C05533=1107.470,43.607,-54.704,179.966,7.215,149.356
C05534=1107.464,43.857,-54.721,179.966,7.219,149.357
C05535=1107.459,44.106,-54.737,179.968,7.222,149.357
C05536=1107.455,44.355,-54.754,179.969,7.227,149.358
C05537=1107.449,44.605,-54.770,179.970,7.231,149.359
C05538=1107.444,44.855,-54.787,179.970,7.235,149.359
C05539=1107.440,45.104,-54.804,179.971,7.239,149.360
C05540=1107.435,45.353,-54.820,179.973,7.243,149.360
C05541=1107.430,45.602,-54.837,179.974,7.247,149.361
C05542=1107.425,45.852,-54.854,179.974,7.251,149.362
C05543=1107.420,46.101,-54.870,179.975,7.255,149.362
C05544=1107.415,46.351,-54.886,179.976,7.259,149.363
C05545=1107.411,46.601,-54.903,179.978,7.263,149.364
C05546=1107.405,46.850,-54.920,179.978,7.267,149.364
C05547=1107.400,47.099,-54.936,179.980,7.271,149.365
C05548=1107.396,47.349,-54.953,179.981,7.275,149.365
C05549=1107.390,47.598,-54.970,179.982,7.279,149.366
C05550=1107.385,47.847,-54.987,179.983,7.283,149.367
C05551=1107.381,48.097,-55.003,179.984,7.287,149.367
C05552=1107.375,48.346,-55.020,179.985,7.291,149.368
C05553=1107.371,48.595,-55.037,179.986,7.295,149.368
C05554=1107.366,48.845,-55.054,179.987,7.299,149.369
C05555=1107.361,49.094,-55.071,179.988,7.303,149.370
C05556=1107.356,49.343,-55.087,179.989,7.307,149.370
C05557=1107.351,49.593,-55.104,179.991,7.311,149.371
C05558=1107.347,49.806,-55.118,179.992,7.314,149.371
C05559=1107.343,50.020,-55.133,179.992,7.318,149.372
C05560=1107.338,50.235,-55.147,179.993,7.321,149.372
C05561=1107.334,50.448,-55.161,179.994,7.325,149.373
C05562=1107.330,50.662,-55.176,179.995,7.328,149.373
C05563=1107.326,50.876,-55.191,179.996,7.332,149.374
C05564=1107.322,51.090,-55.205,179.997,7.335,149.374
C05565=1107.318,51.304,-55.220,179.998,7.339,149.375
C05566=1107.312,51.553,-55.237,179.999,7.342,149.375
C05567=1107.308,51.803,-55.254,180.000,7.346,149.376
C05568=1107.302,52.052,-55.270,-179.999,7.350,149.376
C05569=1107.298,52.301,-55.287,-179.997,7.355,149.377
C05570=1107.293,52.551,-55.304,-179.997,7.358,149.378
C05571=1107.288,52.801,-55.321,-179.995,7.362,149.378
C05572=1107.284,53.050,-55.338,-179.994,7.366,149.379
C05573=1107.278,53.299,-55.355,-179.993,7.370,149.379
C05574=1107.274,53.548,-55.372,-179.992,7.374,149.380
C05575=1107.268,53.798,-55.389,-179.991,7.378,149.381
C05576=1107.264,54.047,-55.406,-179.990,7.382,149.381
C05577=1107.258,54.296,-55.424,-179.989,7.386,149.382
C05578=1107.254,54.545,-55.440,-179.987,7.390,149.382
C05579=1107.249,54.795,-55.458,-179.986,7.394,149.383
C05580=1107.244,55.045,-55.474,-179.985,7.398,149.383
C05581=1107.239,55.294,-55.491,-179.984,7.402,149.384
C05582=1107.235,55.543,-55.509,-179.983,7.406,149.384
C05583=1107.229,55.792,-55.526,-179.981,7.410,149.385
C05584=1107.224,56.042,-55.543,-179.981,7.414,149.386
C05585=1107.220,56.291,-55.560,-179.980,7.418,149.386
C05586=1107.214,56.541,-55.578,-179.978,7.422,149.387
C05587=1107.210,56.790,-55.594,-179.977,7.426,149.387
C05588=1107.205,57.040,-55.612,-179.975,7.430,149.388
C05589=1107.200,57.288,-55.629,-179.975,7.433,149.388
C05590=1107.195,57.538,-55.646,-179.973,7.437,149.389
C05591=1107.190,57.787,-55.664,-179.972,7.442,149.389
C05592=1107.185,58.037,-55.681,-179.971,7.446,149.390
C05593=1107.180,58.287,-55.698,-179.970,7.450,149.391
C05594=1107.176,58.535,-55.715,-179.969,7.453,149.391
C05595=1107.171,58.785,-55.732,-179.968,7.457,149.392
C05596=1107.165,59.035,-55.750,-179.966,7.461,149.392
C05597=1107.161,59.284,-55.767,-179.965,7.465,149.393
C05598=1107.155,59.533,-55.784,-179.963,7.469,149.393
C05599=1107.151,59.782,-55.802,-179.963,7.473,149.394
C05600=1107.146,60.032,-55.819,-179.961,7.477,149.394
C05601=1107.141,60.281,-55.837,-179.960,7.481,149.395
C05602=1107.136,60.531,-55.854,-179.959,7.485,149.395
C05603=1107.132,60.780,-55.871,-179.958,7.489,149.396
C05604=1107.127,61.029,-55.889,-179.956,7.493,149.396
C05605=1107.122,61.278,-55.907,-179.956,7.497,149.397
C05606=1107.117,61.528,-55.923,-179.954,7.501,149.397
C05607=1107.112,61.777,-55.941,-179.953,7.505,149.398
C05608=1107.107,62.027,-55.958,-179.951,7.509,149.399
C05609=1107.102,62.276,-55.976,-179.950,7.513,149.399
C05610=1107.098,62.526,-55.993,-179.949,7.516,149.400
C05611=1107.093,62.775,-56.011,-179.948,7.520,149.400
C05612=1107.087,63.025,-56.028,-179.947,7.524,149.401
C05613=1107.083,63.274,-56.046,-179.945,7.528,149.401
C05614=1107.079,63.487,-56.061,-179.944,7.531,149.402
C05615=1107.074,63.701,-56.076,-179.944,7.535,149.402
C05616=1107.070,63.915,-56.091,-179.942,7.539,149.403
C05617=1107.065,64.129,-56.106,-179.941,7.542,149.403
C05618=1107.062,64.342,-56.121,-179.940,7.545,149.404
C05619=1107.058,64.556,-56.136,-179.939,7.549,149.404
C05620=1107.054,64.770,-56.151,-179.938,7.552,149.404
C05621=1107.049,64.983,-56.167,-179.937,7.555,149.405
C05622=1107.044,65.233,-56.184,-179.935,7.559,149.405
C05623=1107.039,65.482,-56.202,-179.934,7.563,149.406
C05624=1107.035,65.731,-56.219,-179.933,7.567,149.406
C05625=1107.030,65.981,-56.236,-179.931,7.572,149.407
C05626=1107.025,66.230,-56.254,-179.930,7.575,149.407
C05627=1107.020,66.479,-56.272,-179.929,7.579,149.408
C05628=1107.015,66.729,-56.290,-179.928,7.583,149.409
C05629=1107.010,66.978,-56.308,-179.926,7.587,149.409
C05630=1107.006,67.228,-56.325,-179.925,7.591,149.410
C05631=1107.001,67.477,-56.343,-179.924,7.595,149.410
C05632=1106.996,67.726,-56.361,-179.923,7.598,149.411
C05633=1106.991,67.976,-56.379,-179.921,7.602,149.411
C05634=1106.986,68.225,-56.397,-179.920,7.606,149.412
C05635=1106.981,68.474,-56.415,-179.918,7.610,149.412
C05636=1106.976,68.724,-56.433,-179.917,7.615,149.413
C05637=1106.971,68.973,-56.451,-179.916,7.618,149.413
C05638=1106.966,69.223,-56.468,-179.915,7.623,149.414
C05639=1106.961,69.472,-56.486,-179.913,7.627,149.414
C05640=1106.956,69.721,-56.504,-179.912,7.630,149.415
C05641=1106.952,69.970,-56.521,-179.911,7.634,149.415
C05642=1106.947,70.219,-56.539,-179.909,7.638,149.416
C05643=1106.943,70.469,-56.557,-179.908,7.642,149.416
C05644=1106.938,70.718,-56.575,-179.907,7.646,149.417
C05645=1106.933,70.967,-56.593,-179.905,7.650,149.417
C05646=1106.928,71.216,-56.611,-179.904,7.654,149.418
C05647=1106.923,71.466,-56.629,-179.902,7.658,149.418
C05648=1106.918,71.715,-56.647,-179.901,7.661,149.419
C05649=1106.913,71.965,-56.665,-179.900,7.665,149.419
C05650=1106.908,72.214,-56.683,-179.899,7.669,149.420
C05651=1106.904,72.464,-56.701,-179.897,7.673,149.420
C05652=1106.899,72.713,-56.719,-179.896,7.677,149.421
C05653=1106.894,72.962,-56.737,-179.894,7.682,149.421
C05654=1106.889,73.211,-56.755,-179.893,7.685,149.422
C05655=1106.884,73.461,-56.773,-179.891,7.689,149.422
C05656=1106.879,73.710,-56.791,-179.890,7.693,149.423
C05657=1106.874,73.960,-56.810,-179.889,7.697,149.423
C05658=1106.870,74.209,-56.828,-179.888,7.701,149.424
C05659=1106.865,74.458,-56.846,-179.886,7.705,149.424
C05660=1106.860,74.707,-56.864,-179.885,7.709,149.425
C05661=1106.855,74.956,-56.882,-179.883,7.713,149.425
C05662=1106.851,75.206,-56.901,-179.882,7.717,149.426
C05663=1106.846,75.455,-56.919,-179.880,7.721,149.426
C05664=1106.841,75.704,-56.937,-179.879,7.725,149.427
C05665=1106.836,75.953,-56.955,-179.878,7.729,149.427
C05666=1106.830,76.203,-56.973,-179.876,7.733,149.428
C05667=1106.826,76.453,-56.992,-179.875,7.736,149.428
C05668=1106.821,76.701,-57.010,-179.874,7.740,149.429
C05669=1106.817,76.950,-57.028,-179.872,7.744,149.429
C05670=1106.812,77.164,-57.044,-179.871,7.747,149.430
C05671=1106.808,77.378,-57.059,-179.871,7.751,149.430
C05672=1106.804,77.592,-57.075,-179.870,7.754,149.431
C05673=1106.800,77.806,-57.091,-179.869,7.757,149.431
C05674=1106.796,78.019,-57.106,-179.868,7.760,149.432
C05675=1106.792,78.232,-57.122,-179.867,7.763,149.432
C05676=1106.788,78.446,-57.138,-179.867,7.766,149.433
C05677=1106.783,78.660,-57.154,-179.866,7.770,149.433
C05678=1106.779,78.910,-57.172,-179.864,7.773,149.434
C05679=1106.773,79.159,-57.191,-179.864,7.777,149.434
C05680=1106.769,79.408,-57.209,-179.862,7.781,149.435
C05681=1106.764,79.657,-57.228,-179.861,7.784,149.435
C05682=1106.760,79.907,-57.246,-179.860,7.789,149.436
C05683=1106.755,80.156,-57.264,-179.859,7.792,149.436
C05684=1106.749,80.405,-57.282,-179.858,7.796,149.437
C05685=1106.745,80.655,-57.302,-179.857,7.799,149.437
C05686=1106.740,80.904,-57.320,-179.856,7.803,149.438
C05687=1106.735,81.153,-57.338,-179.855,7.807,149.439
C05688=1106.730,81.402,-57.357,-179.854,7.811,149.439
C05689=1106.726,81.652,-57.375,-179.853,7.814,149.440
C05690=1106.721,81.901,-57.393,-179.852,7.818,149.440
C05691=1106.715,82.150,-57.412,-179.851,7.821,149.441
C05692=1106.711,82.400,-57.431,-179.850,7.826,149.441
C05693=1106.706,82.648,-57.449,-179.849,7.829,149.442
C05694=1106.702,82.897,-57.467,-179.848,7.833,149.442
C05695=1106.696,83.148,-57.486,-179.846,7.837,149.443
C05696=1106.692,83.396,-57.505,-179.846,7.840,149.444
C05697=1106.687,83.645,-57.523,-179.844,7.844,149.444
C05698=1106.682,83.895,-57.543,-179.844,7.848,149.445
C05699=1106.677,84.144,-57.561,-179.842,7.852,149.445
C05700=1106.673,84.394,-57.579,-179.841,7.855,149.446
C05701=1106.668,84.643,-57.598,-179.840,7.859,149.446
C05702=1106.663,84.892,-57.616,-179.839,7.863,149.447
C05703=1106.658,85.142,-57.636,-179.838,7.866,149.447
C05704=1106.653,85.391,-57.654,-179.837,7.871,149.448
C05705=1106.648,85.639,-57.673,-179.835,7.875,149.448
C05706=1106.643,85.890,-57.692,-179.834,7.878,149.449
C05707=1106.639,86.138,-57.710,-179.833,7.882,149.449
C05708=1106.635,86.388,-57.729,-179.832,7.885,149.450
C05709=1106.629,86.637,-57.748,-179.831,7.889,149.450
C05710=1106.625,86.885,-57.767,-179.829,7.893,149.451
C05711=1106.620,87.136,-57.786,-179.828,7.896,149.451
C05712=1106.615,87.384,-57.804,-179.827,7.901,149.452
C05713=1106.610,87.634,-57.823,-179.826,7.905,149.452
C05714=1106.605,87.883,-57.842,-179.825,7.908,149.453
C05715=1106.600,88.132,-57.860,-179.823,7.912,149.454
C05716=1106.596,88.382,-57.880,-179.822,7.916,149.454
C05717=1106.591,88.630,-57.898,-179.821,7.919,149.455
C05718=1106.586,88.880,-57.917,-179.820,7.923,149.455
C05719=1106.581,89.129,-57.936,-179.818,7.927,149.455
C05720=1106.577,89.378,-57.956,-179.818,7.931,149.456
C05721=1106.572,89.628,-57.973,-179.816,7.934,149.457
C05722=1106.567,89.877,-57.993,-179.814,7.938,149.457
C05723=1106.562,90.126,-58.012,-179.814,7.942,149.458
C05724=1106.557,90.376,-58.031,-179.812,7.946,149.458
C05725=1106.553,90.624,-58.049,-179.811,7.950,149.459
C05726=1106.548,90.839,-58.066,-179.810,7.953,149.459
C05727=1106.544,91.052,-58.083,-179.809,7.956,149.459
C05728=1106.540,91.266,-58.099,-179.808,7.959,149.460
C05729=1106.536,91.479,-58.114,-179.806,7.963,149.460
C05730=1106.532,91.693,-58.131,-179.805,7.966,149.461
C05731=1106.528,91.906,-58.147,-179.804,7.969,149.461
C05732=1106.523,92.120,-58.164,-179.803,7.972,149.462
C05733=1106.520,92.334,-58.181,-179.802,7.975,149.462
C05734=1106.515,92.582,-58.199,-179.801,7.979,149.462
C05735=1106.510,92.833,-58.218,-179.799,7.983,149.463
C05736=1106.505,93.082,-58.237,-179.798,7.987,149.463
C05737=1106.501,93.331,-58.256,-179.797,7.990,149.464
C05738=1106.495,93.580,-58.276,-179.795,7.994,149.464
C05739=1106.491,93.829,-58.295,-179.794,7.998,149.465
C05740=1106.486,94.078,-58.313,-179.793,8.001,149.465
C05741=1106.481,94.328,-58.333,-179.791,8.005,149.466
C05742=1106.476,94.576,-58.352,-179.790,8.009,149.466
C05743=1106.472,94.826,-58.371,-179.789,8.013,149.467
C05744=1106.466,95.075,-58.391,-179.787,8.017,149.467
C05745=1106.462,95.324,-58.410,-179.786,8.020,149.468
C05746=1106.457,95.573,-58.429,-179.784,8.024,149.468
C05747=1106.452,95.823,-58.449,-179.783,8.028,149.468
C05748=1106.448,96.072,-58.468,-179.781,8.032,149.469
C05749=1106.443,96.321,-58.487,-179.780,8.035,149.469
C05750=1106.438,96.571,-58.506,-179.779,8.039,149.470
C05751=1106.433,96.819,-58.525,-179.777,8.043,149.470
C05752=1106.428,97.069,-58.544,-179.775,8.047,149.471
C05753=1106.424,97.319,-58.564,-179.774,8.051,149.471
C05754=1106.419,97.567,-58.583,-179.773,8.054,149.472
C05755=1106.414,97.817,-58.602,-179.772,8.058,149.472
C05756=1106.409,98.066,-58.622,-179.770,8.062,149.473
C05757=1106.404,98.315,-58.641,-179.768,8.066,149.473
C05758=1106.400,98.564,-58.660,-179.767,8.070,149.474
C05759=1106.395,98.813,-58.680,-179.766,8.073,149.474
C05760=1106.391,99.062,-58.700,-179.764,8.076,149.474
C05761=1106.386,99.312,-58.720,-179.762,8.080,149.475
C05762=1106.381,99.560,-58.738,-179.761,8.084,149.475
C05763=1106.376,99.810,-58.758,-179.759,8.088,149.475
C05764=1106.371,100.059,-58.777,-179.757,8.092,149.476
C05765=1106.366,100.308,-58.797,-179.756,8.095,149.476
C05766=1106.362,100.558,-58.817,-179.755,8.099,149.477
C05767=1106.357,100.807,-58.835,-179.753,8.103,149.477
C05768=1106.352,101.056,-58.855,-179.752,8.107,149.478
C05769=1106.348,101.305,-58.875,-179.750,8.111,149.478
C05770=1106.342,101.554,-58.895,-179.748,8.114,149.478
C05771=1106.338,101.803,-58.914,-179.747,8.117,149.479
C05772=1106.333,102.053,-58.934,-179.745,8.121,149.479
C05773=1106.329,102.302,-58.953,-179.744,8.125,149.480
C05774=1106.324,102.551,-58.973,-179.742,8.129,149.480
C05775=1106.319,102.800,-58.993,-179.740,8.132,149.480
C05776=1106.314,103.050,-59.012,-179.739,8.136,149.481
C05777=1106.309,103.299,-59.032,-179.738,8.139,149.481
C05778=1106.305,103.547,-59.052,-179.736,8.143,149.482
C05779=1106.300,103.797,-59.072,-179.734,8.147,149.482
C05780=1106.295,104.046,-59.091,-179.732,8.151,149.482
C05781=1106.290,104.296,-59.111,-179.731,8.154,149.483
C05782=1106.286,104.509,-59.127,-179.729,8.157,149.483
C05783=1106.282,104.723,-59.145,-179.728,8.161,149.483
C05784=1106.278,104.936,-59.161,-179.726,8.164,149.484
C05785=1106.274,105.149,-59.179,-179.725,8.167,149.484
C05786=1106.270,105.363,-59.196,-179.723,8.170,149.484
C05787=1106.266,105.577,-59.213,-179.722,8.173,149.484
C05788=1106.262,105.791,-59.229,-179.721,8.176,149.485
C05789=1106.257,106.004,-59.246,-179.719,8.179,149.485
C05790=1106.253,106.253,-59.266,-179.718,8.183,149.486
C05791=1106.248,106.502,-59.286,-179.716,8.186,149.486
C05792=1106.244,106.751,-59.306,-179.714,8.190,149.486
C05793=1106.238,107.000,-59.326,-179.712,8.194,149.486
C05794=1106.234,107.250,-59.345,-179.710,8.198,149.487
C05795=1106.229,107.499,-59.366,-179.708,8.201,149.487
C05796=1106.224,107.748,-59.385,-179.707,8.205,149.488
C05797=1106.220,107.997,-59.406,-179.705,8.209,149.488
C05798=1106.215,108.246,-59.425,-179.704,8.212,149.488
C05799=1106.210,108.495,-59.445,-179.702,8.215,149.488
C05800=1106.205,108.744,-59.465,-179.700,8.219,149.489
C05801=1106.201,108.993,-59.486,-179.698,8.222,149.489
C05802=1106.196,109.243,-59.505,-179.696,8.226,149.490
C05803=1106.192,109.492,-59.526,-179.694,8.230,149.490
C05804=1106.186,109.741,-59.545,-179.692,8.233,149.490
C05805=1106.182,109.990,-59.565,-179.691,8.237,149.490
C05806=1106.177,110.239,-59.585,-179.689,8.241,149.491
C05807=1106.172,110.489,-59.606,-179.687,8.244,149.491
C05808=1106.168,110.738,-59.626,-179.685,8.248,149.491
C05809=1106.163,110.987,-59.646,-179.684,8.251,149.492
C05810=1106.159,111.236,-59.666,-179.681,8.254,149.492
C05811=1106.153,111.485,-59.686,-179.680,8.258,149.492
C05812=1106.149,111.734,-59.706,-179.678,8.262,149.492
C05813=1106.144,111.983,-59.726,-179.677,8.265,149.493
C05814=1106.139,112.233,-59.747,-179.675,8.268,149.493
C05815=1106.134,112.482,-59.767,-179.673,8.272,149.493
C05816=1106.130,112.731,-59.787,-179.672,8.275,149.494
C05817=1106.125,112.980,-59.807,-179.670,8.278,149.494
C05818=1106.121,113.229,-59.827,-179.668,8.282,149.494
C05819=1106.116,113.478,-59.848,-179.666,8.286,149.495
C05820=1106.110,113.727,-59.868,-179.665,8.289,149.495
C05821=1106.106,113.976,-59.888,-179.663,8.292,149.495
C05822=1106.101,114.225,-59.908,-179.661,8.296,149.496
C05823=1106.097,114.474,-59.929,-179.659,8.299,149.496
C05824=1106.091,114.724,-59.949,-179.658,8.303,149.496
C05825=1106.087,114.973,-59.969,-179.656,8.306,149.496
C05826=1106.083,115.222,-59.990,-179.654,8.309,149.497
C05827=1106.077,115.471,-60.011,-179.653,8.313,149.497
C05828=1106.073,115.720,-60.031,-179.651,8.316,149.497
C05829=1106.068,115.970,-60.051,-179.649,8.319,149.498
C05830=1106.064,116.219,-60.071,-179.648,8.323,149.498
C05831=1106.059,116.468,-60.092,-179.646,8.326,149.498
C05832=1106.054,116.717,-60.112,-179.644,8.329,149.498
C05833=1106.050,116.966,-60.133,-179.642,8.333,149.499
C05834=1106.045,117.215,-60.154,-179.640,8.336,149.499
C05835=1106.040,117.465,-60.173,-179.639,8.339,149.499
C05836=1106.035,117.714,-60.194,-179.637,8.343,149.500
C05837=1106.030,117.963,-60.215,-179.635,8.346,149.500
C05838=1106.027,118.176,-60.232,-179.634,8.349,149.500
C05839=1106.023,118.389,-60.250,-179.632,8.352,149.500
C05840=1106.019,118.603,-60.268,-179.631,8.355,149.501
C05841=1106.015,118.816,-60.285,-179.630,8.357,149.501
C05842=1106.010,119.030,-60.303,-179.628,8.361,149.501
C05843=1106.006,119.243,-60.320,-179.627,8.364,149.502
C05844=1106.002,119.456,-60.337,-179.625,8.367,149.502
C05845=1105.998,119.669,-60.355,-179.624,8.369,149.502
C05846=1105.993,119.919,-60.376,-179.622,8.373,149.502
C05847=1105.989,120.168,-60.397,-179.620,8.376,149.503
C05848=1105.984,120.417,-60.418,-179.619,8.379,149.503
C05849=1105.980,120.666,-60.438,-179.616,8.383,149.503
C05850=1105.975,120.915,-60.459,-179.615,8.386,149.503
C05851=1105.970,121.165,-60.480,-179.613,8.389,149.504
C05852=1105.966,121.414,-60.500,-179.611,8.393,149.504
C05853=1105.960,121.663,-60.521,-179.610,8.396,149.504
C05854=1105.956,121.912,-60.541,-179.608,8.399,149.505
C05855=1105.951,122.161,-60.562,-179.606,8.403,149.505
C05856=1105.946,122.410,-60.583,-179.605,8.406,149.505
C05857=1105.942,122.659,-60.603,-179.603,8.409,149.505
C05858=1105.937,122.908,-60.625,-179.601,8.413,149.506
C05859=1105.933,123.156,-60.645,-179.600,8.416,149.506
C05860=1105.928,123.406,-60.666,-179.598,8.419,149.506
C05861=1105.924,123.655,-60.687,-179.596,8.423,149.507
C05862=1105.918,123.905,-60.708,-179.593,8.426,149.507
C05863=1105.914,124.154,-60.728,-179.592,8.430,149.507
C05864=1105.909,124.403,-60.749,-179.590,8.433,149.507
C05865=1105.905,124.651,-60.770,-179.588,8.437,149.508
C05866=1105.900,124.900,-60.791,-179.587,8.439,149.508
C05867=1105.894,125.150,-60.812,-179.585,8.443,149.508
C05868=1105.891,125.399,-60.833,-179.583,8.447,149.509
C05869=1105.886,125.648,-60.855,-179.582,8.449,149.509
C05870=1105.881,125.897,-60.875,-179.580,8.453,149.509
C05871=1105.876,126.146,-60.896,-179.578,8.456,149.509
C05872=1105.872,126.395,-60.916,-179.577,8.459,149.510
C05873=1105.867,126.644,-60.938,-179.575,8.463,149.510
C05874=1105.862,126.894,-60.959,-179.572,8.466,149.510
C05875=1105.858,127.143,-60.980,-179.571,8.469,149.510
C05876=1105.853,127.391,-61.001,-179.569,8.473,149.511
C05877=1105.848,127.640,-61.022,-179.567,8.476,149.511
C05878=1105.843,127.890,-61.043,-179.566,8.479,149.511
C05879=1105.839,128.139,-61.065,-179.564,8.483,149.512
C05880=1105.835,128.388,-61.085,-179.562,8.487,149.512
C05881=1105.829,128.637,-61.106,-179.561,8.489,149.512
C05882=1105.825,128.886,-61.128,-179.559,8.493,149.512
C05883=1105.820,129.135,-61.148,-179.557,8.496,149.513
C05884=1105.816,129.384,-61.170,-179.556,8.499,149.513
C05885=1105.811,129.633,-61.191,-179.554,8.503,149.513
C05886=1105.806,129.882,-61.212,-179.552,8.506,149.514
C05887=1105.801,130.131,-61.233,-179.549,8.510,149.514
C05888=1105.796,130.380,-61.254,-179.548,8.513,149.514
C05889=1105.792,130.629,-61.276,-179.546,8.516,149.514
C05890=1105.787,130.878,-61.297,-179.544,8.520,149.515
C05891=1105.783,131.127,-61.318,-179.543,8.523,149.515
C05892=1105.777,131.376,-61.339,-179.541,8.527,149.515
C05893=1105.774,131.625,-61.361,-179.539,8.530,149.516
C05894=1105.769,131.839,-61.379,-179.538,8.533,149.516
C05895=1105.765,132.052,-61.398,-179.536,8.535,149.516
C05896=1105.761,132.265,-61.416,-179.535,8.538,149.516
C05897=1105.757,132.478,-61.434,-179.533,8.541,149.517
C05898=1105.753,132.691,-61.452,-179.531,8.544,149.517
C05899=1105.749,132.906,-61.470,-179.530,8.547,149.517
C05900=1105.745,133.119,-61.488,-179.528,8.550,149.517
C05901=1105.741,133.332,-61.507,-179.527,8.553,149.518
C05902=1105.736,133.581,-61.528,-179.525,8.556,149.518
C05903=1105.731,133.830,-61.550,-179.524,8.559,149.518
C05904=1105.728,134.080,-61.571,-179.522,8.563,149.518
C05905=1105.723,134.328,-61.592,-179.520,8.566,149.519
C05906=1105.718,134.577,-61.614,-179.518,8.570,149.519
C05907=1105.713,134.827,-61.635,-179.517,8.573,149.519
C05908=1105.708,135.075,-61.657,-179.515,8.576,149.519
C05909=1105.704,135.324,-61.679,-179.513,8.580,149.520
C05910=1105.700,135.574,-61.699,-179.512,8.583,149.520
C05911=1105.695,135.822,-61.721,-179.510,8.586,149.520
C05912=1105.690,136.071,-61.743,-179.508,8.590,149.521
C05913=1105.685,136.321,-61.764,-179.506,8.594,149.521
C05914=1105.681,136.570,-61.786,-179.504,8.596,149.521
C05915=1105.676,136.818,-61.808,-179.502,8.600,149.522
C05916=1105.671,137.068,-61.830,-179.501,8.604,149.522
C05917=1105.666,137.317,-61.851,-179.499,8.606,149.522
C05918=1105.662,137.566,-61.873,-179.497,8.610,149.522
C05919=1105.658,137.814,-61.894,-179.496,8.614,149.523
C05920=1105.653,138.063,-61.915,-179.493,8.617,149.523
C05921=1105.648,138.313,-61.937,-179.492,8.620,149.523
C05922=1105.643,138.562,-61.958,-179.490,8.624,149.524
C05923=1105.639,138.811,-61.980,-179.488,8.627,149.524
C05924=1105.634,139.060,-62.002,-179.486,8.631,149.524
C05925=1105.629,139.308,-62.024,-179.485,8.634,149.525
C05926=1105.625,139.558,-62.046,-179.483,8.637,149.525
C05927=1105.620,139.806,-62.068,-179.481,8.641,149.525
C05928=1105.616,140.056,-62.089,-179.479,8.645,149.526
C05929=1105.611,140.305,-62.111,-179.478,8.647,149.526
C05930=1105.607,140.554,-62.133,-179.476,8.651,149.526
C05931=1105.602,140.803,-62.154,-179.474,8.655,149.527
C05932=1105.597,141.052,-62.176,-179.472,8.658,149.527
C05933=1105.593,141.301,-62.198,-179.471,8.661,149.527
C05934=1105.588,141.550,-62.220,-179.469,8.665,149.527
C05935=1105.583,141.799,-62.242,-179.467,8.668,149.528
C05936=1105.579,142.048,-62.263,-179.465,8.672,149.528
C05937=1105.574,142.297,-62.285,-179.464,8.675,149.528
C05938=1105.569,142.545,-62.307,-179.462,8.678,149.529
C05939=1105.565,142.795,-62.329,-179.460,8.682,149.529
C05940=1105.560,143.043,-62.351,-179.458,8.686,149.529
C05941=1105.555,143.293,-62.374,-179.457,8.689,149.530
C05942=1105.550,143.542,-62.395,-179.455,8.692,149.530
C05943=1105.546,143.791,-62.417,-179.453,8.696,149.530
C05944=1105.541,144.040,-62.439,-179.451,8.700,149.531
C05945=1105.537,144.289,-62.461,-179.449,8.703,149.531
C05946=1105.532,144.538,-62.483,-179.448,8.706,149.531
C05947=1105.528,144.787,-62.505,-179.446,8.710,149.532
C05948=1105.523,145.036,-62.526,-179.445,8.714,149.532
C05949=1105.518,145.285,-62.550,-179.442,8.717,149.532
C05950=1105.514,145.498,-62.568,-179.441,8.720,149.532
C05951=1105.510,145.711,-62.587,-179.440,8.723,149.533
C05952=1105.507,145.925,-62.606,-179.438,8.726,149.533
C05953=1105.502,146.137,-62.625,-179.436,8.729,149.533
C05954=1105.498,146.351,-62.643,-179.435,8.732,149.534
C05955=1105.495,146.564,-62.663,-179.433,8.735,149.534
C05956=1105.491,146.777,-62.681,-179.432,8.738,149.534
C05957=1105.486,146.990,-62.701,-179.430,8.741,149.534
C05958=1105.482,147.240,-62.723,-179.428,8.745,149.535
C05959=1105.478,147.489,-62.745,-179.426,8.748,149.535
C05960=1105.473,147.737,-62.767,-179.424,8.752,149.535
C05961=1105.468,147.987,-62.790,-179.423,8.754,149.535
C05962=1105.463,148.235,-62.812,-179.421,8.758,149.536
C05963=1105.459,148.485,-62.834,-179.419,8.762,149.536
C05964=1105.455,148.733,-62.856,-179.417,8.765,149.536
C05965=1105.449,148.982,-62.879,-179.415,8.769,149.537
C05966=1105.445,149.232,-62.901,-179.413,8.771,149.537
C05967=1105.440,149.480,-62.922,-179.412,8.775,149.537
C05968=1105.436,149.729,-62.945,-179.410,8.779,149.537
C05969=1105.431,149.979,-62.968,-179.408,8.782,149.538
C05970=1105.426,150.227,-62.989,-179.406,8.786,149.538
C05971=1105.423,150.476,-63.012,-179.404,8.788,149.538
C05972=1105.417,150.725,-63.034,-179.402,8.792,149.538
C05973=1105.413,150.974,-63.057,-179.400,8.795,149.539
C05974=1105.409,151.223,-63.079,-179.398,8.799,149.539
C05975=1105.403,151.472,-63.102,-179.396,8.802,149.539
C05976=1105.399,151.721,-63.124,-179.394,8.805,149.539
C05977=1105.395,151.970,-63.146,-179.392,8.809,149.540
C05978=1105.390,152.218,-63.169,-179.390,8.812,149.540
C05979=1105.385,152.468,-63.191,-179.388,8.816,149.540
C05980=1105.381,152.717,-63.215,-179.387,8.818,149.540
C05981=1105.376,152.965,-63.236,-179.385,8.822,149.541
C05982=1105.371,153.215,-63.259,-179.383,8.825,149.541
C05983=1105.367,153.464,-63.282,-179.380,8.829,149.541
C05984=1105.362,153.712,-63.304,-179.379,8.831,149.541
C05985=1105.357,153.961,-63.327,-179.377,8.835,149.542
C05986=1105.353,154.210,-63.350,-179.375,8.838,149.542
C05987=1105.348,154.459,-63.372,-179.373,8.841,149.542
C05988=1105.344,154.708,-63.395,-179.371,8.845,149.542
C05989=1105.339,154.957,-63.417,-179.369,8.848,149.542
C05990=1105.335,155.206,-63.440,-179.367,8.852,149.543
C05991=1105.330,155.455,-63.462,-179.365,8.854,149.543
C05992=1105.325,155.704,-63.485,-179.363,8.857,149.543
C05993=1105.321,155.953,-63.508,-179.361,8.861,149.543
C05994=1105.316,156.202,-63.531,-179.359,8.864,149.543
C05995=1105.312,156.450,-63.553,-179.358,8.867,149.544
C05996=1105.307,156.700,-63.576,-179.355,8.870,149.544
C05997=1105.303,156.949,-63.598,-179.353,8.874,149.544
C05998=1105.298,157.198,-63.622,-179.351,8.876,149.544
C05999=1105.293,157.446,-63.643,-179.349,8.880,149.544
C06000=1105.288,157.695,-63.667,-179.347,8.883,149.544
C06001=1105.284,157.944,-63.690,-179.345,8.886,149.545
C06002=1105.280,158.193,-63.713,-179.343,8.889,149.545
C06003=1105.274,158.442,-63.735,-179.341,8.893,149.545
C06004=1105.270,158.691,-63.758,-179.339,8.896,149.545
C06005=1105.265,158.940,-63.781,-179.337,8.899,149.545
C06006=1105.262,159.153,-63.801,-179.336,8.901,149.546
C06007=1105.258,159.366,-63.820,-179.333,8.904,149.546
C06008=1105.254,159.579,-63.840,-179.332,8.907,149.546
C06009=1105.250,159.792,-63.859,-179.330,8.909,149.546
C06010=1105.246,160.006,-63.879,-179.329,8.912,149.546
C06011=1105.242,160.219,-63.898,-179.327,8.914,149.546
C06012=1105.238,160.432,-63.918,-179.325,8.917,149.546
C06013=1105.235,160.644,-63.938,-179.323,8.919,149.547
C06014=1105.230,160.894,-63.960,-179.321,8.923,149.547
C06015=1105.225,161.143,-63.984,-179.319,8.926,149.547
C06016=1105.221,161.392,-64.007,-179.317,8.929,149.547
C06017=1105.216,161.641,-64.030,-179.315,8.932,149.547
C06018=1105.212,161.890,-64.053,-179.313,8.935,149.547
C06019=1105.207,162.138,-64.076,-179.311,8.938,149.548
C06020=1105.202,162.387,-64.099,-179.309,8.942,149.548
C06021=1105.198,162.636,-64.122,-179.307,8.945,149.548
C06022=1105.194,162.884,-64.145,-179.305,8.947,149.548
C06023=1105.189,163.133,-64.169,-179.303,8.950,149.548
C06024=1105.184,163.382,-64.192,-179.301,8.954,149.548
C06025=1105.180,163.632,-64.214,-179.299,8.956,149.548
C06026=1105.175,163.881,-64.237,-179.297,8.960,149.549
C06027=1105.170,164.129,-64.260,-179.294,8.963,149.549
C06028=1105.165,164.378,-64.284,-179.293,8.966,149.549
C06029=1105.161,164.627,-64.306,-179.290,8.969,149.549
C06030=1105.157,164.876,-64.330,-179.288,8.972,149.549
C06031=1105.152,165.124,-64.354,-179.286,8.975,149.549
C06032=1105.147,165.373,-64.377,-179.284,8.978,149.549
C06033=1105.144,165.622,-64.400,-179.281,8.981,149.549
C06034=1105.139,165.871,-64.423,-179.280,8.984,149.550
C06035=1105.134,166.120,-64.447,-179.277,8.987,149.550
C06036=1105.129,166.369,-64.470,-179.275,8.990,149.550
C06037=1105.125,166.618,-64.493,-179.274,8.993,149.550
C06038=1105.121,166.867,-64.516,-179.271,8.996,149.550
C06039=1105.116,167.116,-64.540,-179.269,8.999,149.550
C06040=1105.111,167.365,-64.563,-179.267,9.002,149.550
C06041=1105.106,167.613,-64.586,-179.265,9.005,149.551
C06042=1105.102,167.862,-64.610,-179.262,9.008,149.551
C06043=1105.097,168.111,-64.633,-179.261,9.011,149.551
C06044=1105.092,168.360,-64.657,-179.258,9.014,149.551
C06045=1105.088,168.609,-64.679,-179.257,9.017,149.551
C06046=1105.084,168.858,-64.703,-179.254,9.020,149.551
C06047=1105.079,169.106,-64.727,-179.252,9.023,149.551
C06048=1105.075,169.355,-64.750,-179.250,9.026,149.551
C06049=1105.070,169.604,-64.774,-179.248,9.029,149.552
C06050=1105.065,169.853,-64.797,-179.246,9.032,149.552
C06051=1105.061,170.101,-64.821,-179.244,9.035,149.552
C06052=1105.056,170.351,-64.844,-179.241,9.038,149.552
C06053=1105.051,170.600,-64.868,-179.239,9.041,149.552
C06054=1105.047,170.849,-64.891,-179.237,9.044,149.552
C06055=1105.042,171.097,-64.915,-179.235,9.047,149.552
C06056=1105.038,171.347,-64.939,-179.233,9.049,149.552
C06057=1105.033,171.596,-64.962,-179.231,9.053,149.552
C06058=1105.029,171.844,-64.986,-179.228,9.056,149.552
C06059=1105.024,172.093,-65.010,-179.227,9.058,149.553
C06060=1105.020,172.342,-65.034,-179.224,9.061,149.553
C06061=1105.015,172.591,-65.057,-179.222,9.065,149.553
C06062=1105.008,173.002,-65.096,-179.219,9.070,149.553
C06063=1105.001,173.414,-65.135,-179.215,9.075,149.553
C06064=1104.993,173.826,-65.174,-179.211,9.079,149.553
C06065=1104.986,174.238,-65.213,-179.208,9.084,149.554
C06066=1104.752,164.026,-64.305,-179.293,8.963,149.548
C06067=1104.756,163.778,-64.282,-179.295,8.960,149.548
C06068=1104.761,163.529,-64.259,-179.297,8.956,149.548
C06069=1104.766,163.280,-64.236,-179.299,8.954,149.548
C06070=1104.770,163.032,-64.213,-179.301,8.951,149.548
C06071=1104.775,162.783,-64.190,-179.303,8.948,149.548
C06072=1104.780,162.534,-64.166,-179.305,8.945,149.547
C06073=1104.784,162.284,-64.144,-179.308,8.942,149.547
C06074=1104.788,162.035,-64.121,-179.309,8.939,149.547
C06075=1104.793,161.786,-64.098,-179.312,8.936,149.547
C06076=1104.797,161.537,-64.075,-179.314,8.932,149.547
C06077=1104.802,161.289,-64.052,-179.315,8.930,149.547
C06078=1104.807,161.040,-64.029,-179.318,8.926,149.547
C06079=1104.811,160.791,-64.006,-179.320,8.923,149.546
C06080=1104.816,160.542,-63.982,-179.321,8.920,149.546
C06081=1104.821,160.293,-63.960,-179.324,8.917,149.546
C06082=1104.825,160.044,-63.937,-179.326,8.914,149.546
C06083=1104.830,159.769,-63.912,-179.328,8.910,149.546
C06084=1104.835,159.494,-63.886,-179.330,8.907,149.546
C06085=1104.840,159.219,-63.861,-179.332,8.904,149.545
C06086=1104.845,158.944,-63.835,-179.335,8.900,149.545
C06087=1104.849,158.695,-63.813,-179.337,8.897,149.545
C06088=1104.855,158.447,-63.790,-179.339,8.894,149.545
C06089=1104.859,158.197,-63.768,-179.341,8.891,149.545
C06090=1104.864,157.948,-63.744,-179.343,8.887,149.544
C06091=1104.868,157.699,-63.721,-179.345,8.885,149.544
C06092=1104.873,157.450,-63.699,-179.347,8.881,149.544
C06093=1104.878,157.202,-63.676,-179.349,8.878,149.544
C06094=1104.882,156.953,-63.653,-179.351,8.875,149.544
C06095=1104.887,156.703,-63.630,-179.353,8.872,149.544
C06096=1104.891,156.454,-63.608,-179.355,8.869,149.543
C06097=1104.896,156.206,-63.585,-179.357,8.865,149.543
C06098=1104.900,155.957,-63.563,-179.358,8.862,149.543
C06099=1104.905,155.708,-63.539,-179.360,8.859,149.543
C06100=1104.909,155.459,-63.517,-179.362,8.856,149.542
C06101=1104.915,155.210,-63.494,-179.364,8.853,149.542
C06102=1104.919,154.961,-63.472,-179.366,8.850,149.542
C06103=1104.924,154.712,-63.449,-179.369,8.846,149.542
C06104=1104.928,154.463,-63.426,-179.371,8.843,149.542
C06105=1104.932,154.215,-63.404,-179.372,8.840,149.541
C06106=1104.937,153.965,-63.381,-179.374,8.837,149.541
C06107=1104.941,153.717,-63.358,-179.376,8.833,149.541
C06108=1104.947,153.468,-63.336,-179.378,8.830,149.541
C06109=1104.951,153.219,-63.313,-179.380,8.827,149.540
C06110=1104.956,152.969,-63.291,-179.382,8.823,149.540
C06111=1104.960,152.721,-63.268,-179.384,8.820,149.540
C06112=1104.964,152.472,-63.246,-179.385,8.817,149.540
C06113=1104.969,152.223,-63.223,-179.387,8.814,149.539
C06114=1104.974,151.974,-63.201,-179.390,8.810,149.539
C06115=1104.979,151.725,-63.178,-179.392,8.807,149.539
C06116=1104.983,151.476,-63.156,-179.393,8.804,149.539
C06117=1104.988,151.227,-63.134,-179.395,8.800,149.539
C06118=1104.993,150.978,-63.111,-179.397,8.797,149.538
C06119=1104.997,150.729,-63.089,-179.399,8.794,149.538
C06120=1105.002,150.480,-63.067,-179.401,8.791,149.538
C06121=1105.006,150.231,-63.044,-179.403,8.787,149.538
C06122=1105.011,149.982,-63.022,-179.405,8.784,149.537
C06123=1105.016,149.733,-63.000,-179.407,8.780,149.537
C06124=1105.020,149.484,-62.977,-179.409,8.777,149.537
C06125=1105.025,149.236,-62.955,-179.410,8.774,149.536
C06126=1105.029,148.986,-62.933,-179.412,8.770,149.536
C06127=1105.033,148.737,-62.910,-179.414,8.767,149.536
C06128=1105.039,148.489,-62.888,-179.416,8.763,149.536
C06129=1105.043,148.239,-62.866,-179.418,8.761,149.535
C06130=1105.048,147.991,-62.843,-179.419,8.757,149.535
C06131=1105.052,147.742,-62.821,-179.422,8.753,149.535
C06132=1105.057,147.492,-62.799,-179.424,8.750,149.535
C06133=1105.062,147.244,-62.777,-179.425,8.746,149.534
C06134=1105.066,146.995,-62.754,-179.427,8.742,149.534
C06135=1105.071,146.781,-62.735,-179.429,8.740,149.534
C06136=1105.074,146.569,-62.717,-179.430,8.737,149.533
C06137=1105.078,146.355,-62.698,-179.432,8.734,149.533
C06138=1105.082,146.142,-62.679,-179.434,8.731,149.533
C06139=1105.087,145.929,-62.660,-179.435,8.728,149.533
C06140=1105.090,145.715,-62.641,-179.436,8.725,149.532
C06141=1105.094,145.502,-62.622,-179.438,8.722,149.532
C06142=1105.098,145.289,-62.603,-179.440,8.719,149.532
C06143=1105.102,145.040,-62.581,-179.441,8.715,149.531
C06144=1105.108,144.791,-62.559,-179.443,8.712,149.531
C06145=1105.112,144.542,-62.537,-179.444,8.708,149.531
C06146=1105.117,144.293,-62.515,-179.447,8.705,149.530
C06147=1105.121,144.044,-62.492,-179.449,8.701,149.530
C06148=1105.126,143.796,-62.471,-179.450,8.697,149.530
C06149=1105.130,143.546,-62.449,-179.452,8.695,149.530
C06150=1105.135,143.298,-62.427,-179.453,8.691,149.529
C06151=1105.139,143.048,-62.405,-179.455,8.687,149.529
C06152=1105.144,142.800,-62.383,-179.457,8.684,149.529
C06153=1105.149,142.550,-62.361,-179.458,8.681,149.528
C06154=1105.154,142.301,-62.339,-179.461,8.677,149.528
C06155=1105.158,142.052,-62.317,-179.462,8.673,149.528
C06156=1105.163,141.803,-62.295,-179.464,8.670,149.527
C06157=1105.167,141.554,-62.273,-179.466,8.666,149.527
C06158=1105.172,141.306,-62.251,-179.467,8.663,149.527
C06159=1105.176,141.056,-62.229,-179.469,8.660,149.526
C06160=1105.181,140.808,-62.208,-179.472,8.656,149.526
C06161=1105.186,140.558,-62.186,-179.473,8.653,149.526
C06162=1105.190,140.310,-62.164,-179.475,8.650,149.525
C06163=1105.196,140.060,-62.143,-179.476,8.646,149.525
C06164=1105.200,139.811,-62.121,-179.478,8.642,149.525
C06165=1105.205,139.562,-62.099,-179.480,8.639,149.525
C06166=1105.209,139.313,-62.077,-179.481,8.636,149.524
C06167=1105.214,139.064,-62.056,-179.483,8.632,149.524
C06168=1105.218,138.815,-62.033,-179.486,8.629,149.524
C06169=1105.223,138.566,-62.012,-179.487,8.625,149.523
C06170=1105.228,138.317,-61.991,-179.489,8.622,149.523
C06171=1105.233,138.068,-61.969,-179.491,8.619,149.523
C06172=1105.237,137.819,-61.947,-179.492,8.615,149.522
C06173=1105.241,137.570,-61.926,-179.494,8.612,149.522
C06174=1105.246,137.321,-61.904,-179.496,8.609,149.522
C06175=1105.251,137.072,-61.883,-179.498,8.605,149.522
C06176=1105.255,136.823,-61.861,-179.500,8.601,149.521
C06177=1105.260,136.574,-61.839,-179.501,8.599,149.521
C06178=1105.265,136.326,-61.818,-179.503,8.595,149.521
C06179=1105.270,136.076,-61.796,-179.505,8.591,149.520
C06180=1105.274,135.827,-61.775,-179.507,8.588,149.520
C06181=1105.279,135.578,-61.753,-179.508,8.585,149.520
C06182=1105.284,135.329,-61.731,-179.510,8.582,149.520
C06183=1105.288,135.080,-61.710,-179.512,8.578,149.519
C06184=1105.292,134.831,-61.688,-179.513,8.575,149.519
C06185=1105.297,134.582,-61.667,-179.515,8.572,149.519
C06186=1105.302,134.333,-61.646,-179.517,8.568,149.518
C06187=1105.307,134.083,-61.624,-179.519,8.564,149.518
C06188=1105.312,133.834,-61.603,-179.521,8.561,149.518
C06189=1105.316,133.586,-61.582,-179.523,8.558,149.517
C06190=1105.321,133.337,-61.560,-179.524,8.554,149.517
C06191=1105.324,133.123,-61.541,-179.526,8.551,149.517
C06192=1105.329,132.910,-61.523,-179.527,8.549,149.517
C06193=1105.333,132.697,-61.505,-179.529,8.546,149.516
C06194=1105.337,132.484,-61.487,-179.530,8.543,149.516
C06195=1105.341,132.270,-61.468,-179.532,8.540,149.516
C06196=1105.345,132.057,-61.450,-179.534,8.537,149.516
C06197=1105.348,131.844,-61.432,-179.535,8.534,149.515
C06198=1105.353,131.630,-61.413,-179.536,8.532,149.515
C06199=1105.357,131.381,-61.393,-179.538,8.528,149.515
C06200=1105.362,131.132,-61.371,-179.539,8.525,149.515
C06201=1105.367,130.883,-61.350,-179.542,8.522,149.514
C06202=1105.371,130.634,-61.328,-179.544,8.518,149.514
C06203=1105.376,130.385,-61.308,-179.545,8.514,149.514
C06204=1105.381,130.136,-61.286,-179.547,8.511,149.513
C06205=1105.386,129.887,-61.265,-179.549,8.508,149.513
C06206=1105.390,129.639,-61.244,-179.551,8.504,149.513
C06207=1105.395,129.389,-61.223,-179.552,8.502,149.513
C06208=1105.400,129.139,-61.202,-179.554,8.498,149.512
C06209=1105.405,128.891,-61.180,-179.556,8.494,149.512
C06210=1105.409,128.642,-61.160,-179.557,8.492,149.512
C06211=1105.413,128.392,-61.137,-179.559,8.488,149.512
C06212=1105.418,128.143,-61.117,-179.561,8.484,149.511
C06213=1105.423,127.894,-61.096,-179.563,8.482,149.511
C06214=1105.428,127.646,-61.074,-179.565,8.478,149.511
C06215=1105.433,127.396,-61.053,-179.567,8.475,149.510
C06216=1105.437,127.147,-61.033,-179.568,8.471,149.510
C06217=1105.442,126.898,-61.011,-179.570,8.468,149.510
C06218=1105.446,126.649,-60.991,-179.572,8.464,149.510
C06219=1105.451,126.400,-60.970,-179.573,8.462,149.509
C06220=1105.456,126.151,-60.948,-179.575,8.458,149.509
C06221=1105.461,125.902,-60.928,-179.577,8.454,149.509
C06222=1105.465,125.652,-60.906,-179.579,8.451,149.508
C06223=1105.470,125.403,-60.886,-179.580,8.448,149.508
C06224=1105.474,125.155,-60.864,-179.582,8.444,149.508
C06225=1105.479,124.906,-60.844,-179.584,8.441,149.508
C06226=1105.484,124.656,-60.823,-179.586,8.438,149.507
C06227=1105.488,124.407,-60.803,-179.588,8.435,149.507
C06228=1105.494,124.158,-60.782,-179.589,8.431,149.507
C06229=1105.497,123.909,-60.760,-179.591,8.428,149.506
C06230=1105.502,123.660,-60.739,-179.593,8.425,149.506
C06231=1105.507,123.411,-60.719,-179.595,8.421,149.506
C06232=1105.512,123.162,-60.698,-179.596,8.418,149.505
C06233=1105.516,122.913,-60.677,-179.598,8.414,149.505
C06234=1105.522,122.663,-60.657,-179.600,8.411,149.505
C06235=1105.526,122.415,-60.635,-179.601,8.408,149.505
C06236=1105.531,122.166,-60.614,-179.603,8.404,149.504
C06237=1105.535,121.917,-60.594,-179.605,8.401,149.504
C06238=1105.540,121.667,-60.573,-179.607,8.398,149.504
C06239=1105.544,121.418,-60.552,-179.609,8.395,149.504
C06240=1105.549,121.169,-60.531,-179.610,8.391,149.503
C06241=1105.554,120.920,-60.511,-179.612,8.388,149.503
C06242=1105.559,120.671,-60.490,-179.614,8.385,149.503
C06243=1105.564,120.422,-60.470,-179.615,8.381,149.502
C06244=1105.568,120.173,-60.449,-179.617,8.378,149.502
C06245=1105.573,119.923,-60.428,-179.619,8.374,149.502
C06246=1105.578,119.674,-60.408,-179.621,8.371,149.502
C06247=1105.582,119.461,-60.390,-179.622,8.368,149.501
C06248=1105.586,119.248,-60.372,-179.623,8.365,149.501
C06249=1105.590,119.034,-60.354,-179.625,8.362,149.501
C06250=1105.594,118.821,-60.337,-179.626,8.360,149.501
C06251=1105.597,118.608,-60.319,-179.628,8.357,149.500
C06252=1105.601,118.394,-60.302,-179.630,8.353,149.500
C06253=1105.606,118.180,-60.285,-179.631,8.351,149.500
C06254=1105.610,117.967,-60.266,-179.633,8.348,149.500
C06255=1105.614,117.718,-60.246,-179.634,8.344,149.499
C06256=1105.619,117.469,-60.225,-179.636,8.341,149.499
C06257=1105.624,117.220,-60.205,-179.638,8.338,149.499
C06258=1105.628,116.970,-60.185,-179.640,8.334,149.499
C06259=1105.634,116.721,-60.164,-179.641,8.331,149.498
C06260=1105.638,116.472,-60.144,-179.643,8.328,149.498
C06261=1105.642,116.223,-60.123,-179.645,8.324,149.498
C06262=1105.647,115.974,-60.103,-179.646,8.321,149.497
C06263=1105.653,115.726,-60.082,-179.648,8.318,149.497
C06264=1105.657,115.477,-60.062,-179.650,8.314,149.497
C06265=1105.662,115.227,-60.042,-179.651,8.311,149.496
C06266=1105.667,114.978,-60.021,-179.653,8.308,149.496
C06267=1105.671,114.729,-60.001,-179.655,8.304,149.496
C06268=1105.676,114.480,-59.981,-179.656,8.301,149.495
C06269=1105.681,114.230,-59.961,-179.658,8.298,149.495
C06270=1105.686,113.981,-59.940,-179.660,8.294,149.495
C06271=1105.690,113.732,-59.920,-179.661,8.291,149.494
C06272=1105.695,113.483,-59.899,-179.663,8.287,149.494
C06273=1105.699,113.234,-59.880,-179.665,8.284,149.494
C06274=1105.704,112.985,-59.859,-179.666,8.281,149.494
C06275=1105.709,112.735,-59.838,-179.668,8.277,149.493
C06276=1105.714,112.486,-59.819,-179.670,8.273,149.493
C06277=1105.719,112.238,-59.799,-179.672,8.270,149.493
C06278=1105.723,111.989,-59.778,-179.673,8.267,149.492
C06279=1105.728,111.739,-59.759,-179.675,8.263,149.492
C06280=1105.733,111.490,-59.738,-179.677,8.260,149.492
C06281=1105.738,111.241,-59.717,-179.678,8.257,149.491
C06282=1105.742,110.991,-59.698,-179.680,8.253,149.491
C06283=1105.747,110.742,-59.677,-179.682,8.250,149.491
C06284=1105.751,110.493,-59.657,-179.684,8.246,149.490
C06285=1105.757,110.245,-59.638,-179.686,8.242,149.490
C06286=1105.761,109.996,-59.617,-179.688,8.239,149.490
C06287=1105.767,109.746,-59.597,-179.690,8.235,149.490
C06288=1105.771,109.497,-59.577,-179.692,8.231,149.489
C06289=1105.776,109.247,-59.557,-179.693,8.228,149.489
C06290=1105.780,108.998,-59.537,-179.695,8.225,149.489
C06291=1105.785,108.749,-59.517,-179.697,8.221,149.488
C06292=1105.790,108.500,-59.497,-179.698,8.217,149.488
C06293=1105.795,108.251,-59.477,-179.700,8.214,149.488
C06294=1105.799,108.002,-59.457,-179.702,8.210,149.487
C06295=1105.804,107.752,-59.437,-179.704,8.207,149.487
C06296=1105.808,107.503,-59.417,-179.706,8.203,149.487
C06297=1105.814,107.255,-59.398,-179.707,8.200,149.486
C06298=1105.818,107.006,-59.377,-179.709,8.196,149.486
C06299=1105.823,106.756,-59.358,-179.710,8.192,149.486
C06300=1105.827,106.507,-59.337,-179.712,8.189,149.485
C06301=1105.832,106.258,-59.317,-179.714,8.185,149.485
C06302=1105.837,106.009,-59.298,-179.716,8.181,149.485
C06303=1105.842,105.795,-59.281,-179.717,8.178,149.484
C06304=1105.845,105.581,-59.264,-179.718,8.175,149.484
C06305=1105.849,105.368,-59.247,-179.720,8.172,149.484
C06306=1105.853,105.155,-59.230,-179.721,8.169,149.483
C06307=1105.858,104.941,-59.213,-179.723,8.166,149.483
C06308=1105.861,104.728,-59.196,-179.724,8.162,149.483
C06309=1105.865,104.514,-59.178,-179.726,8.160,149.483
C06310=1105.870,104.301,-59.162,-179.727,8.156,149.482
C06311=1105.874,104.051,-59.142,-179.729,8.153,149.482
C06312=1105.879,103.802,-59.123,-179.731,8.149,149.481
C06313=1105.884,103.552,-59.103,-179.732,8.145,149.481
C06314=1105.889,103.304,-59.083,-179.734,8.142,149.481
C06315=1105.894,103.055,-59.063,-179.736,8.138,149.480
C06316=1105.898,102.805,-59.044,-179.737,8.135,149.480
C06317=1105.904,102.556,-59.024,-179.738,8.131,149.479
C06318=1105.907,102.307,-59.005,-179.740,8.127,149.479
C06319=1105.912,102.058,-58.985,-179.742,8.123,149.479
C06320=1105.917,101.808,-58.965,-179.744,8.120,149.478
C06321=1105.922,101.559,-58.946,-179.745,8.116,149.478
C06322=1105.927,101.310,-58.926,-179.746,8.113,149.477
C06323=1105.931,101.061,-58.906,-179.748,8.109,149.477
C06324=1105.937,100.812,-58.887,-179.749,8.105,149.477
C06325=1105.941,100.563,-58.868,-179.751,8.101,149.476
C06326=1105.945,100.313,-58.848,-179.753,8.097,149.476
C06327=1105.951,100.064,-58.829,-179.755,8.093,149.476
C06328=1105.956,99.815,-58.809,-179.756,8.090,149.475
C06329=1105.960,99.565,-58.789,-179.757,8.087,149.475
C06330=1105.965,99.317,-58.770,-179.759,8.083,149.474
C06331=1105.969,99.068,-58.750,-179.760,8.079,149.474
C06332=1105.975,98.819,-58.731,-179.762,8.075,149.473
C06333=1105.979,98.569,-58.711,-179.763,8.072,149.473
C06334=1105.983,98.320,-58.692,-179.765,8.068,149.472
C06335=1105.989,98.071,-58.673,-179.766,8.064,149.472
C06336=1105.994,97.822,-58.653,-179.768,8.060,149.472
C06337=1105.998,97.572,-58.634,-179.769,8.056,149.471
C06338=1106.003,97.323,-58.615,-179.770,8.053,149.471
C06339=1106.008,97.074,-58.595,-179.772,8.049,149.470
C06340=1106.013,96.825,-58.576,-179.774,8.045,149.470
C06341=1106.018,96.575,-58.556,-179.775,8.041,149.469
C06342=1106.022,96.326,-58.537,-179.777,8.038,149.469
C06343=1106.027,96.077,-58.518,-179.777,8.034,149.468
C06344=1106.032,95.828,-58.498,-179.779,8.030,149.468
C06345=1106.036,95.579,-58.480,-179.781,8.026,149.467
C06346=1106.041,95.330,-58.460,-179.782,8.022,149.467
C06347=1106.046,95.081,-58.441,-179.783,8.019,149.467
C06348=1106.051,94.831,-58.422,-179.785,8.015,149.466
C06349=1106.056,94.581,-58.403,-179.786,8.011,149.466
C06350=1106.061,94.332,-58.384,-179.788,8.008,149.465
C06351=1106.065,94.083,-58.364,-179.788,8.004,149.465
C06352=1106.070,93.834,-58.345,-179.790,8.000,149.464
C06353=1106.074,93.585,-58.326,-179.792,7.996,149.464
C06354=1106.080,93.336,-58.307,-179.793,7.992,149.463
C06355=1106.085,93.086,-58.288,-179.794,7.989,149.463
C06356=1106.089,92.837,-58.269,-179.795,7.985,149.462
C06357=1106.094,92.588,-58.250,-179.797,7.981,149.462
C06358=1106.099,92.339,-58.231,-179.799,7.977,149.461
C06359=1106.103,92.125,-58.214,-179.799,7.974,149.461
C06360=1106.107,91.911,-58.197,-179.800,7.971,149.460
C06361=1106.111,91.698,-58.182,-179.801,7.968,149.460
C06362=1106.115,91.484,-58.165,-179.802,7.965,149.460
C06363=1106.119,91.271,-58.149,-179.803,7.962,149.459
C06364=1106.124,91.057,-58.132,-179.805,7.958,149.459
C06365=1106.128,90.844,-58.116,-179.806,7.955,149.458
C06366=1106.132,90.630,-58.100,-179.807,7.952,149.458
C06367=1106.136,90.381,-58.081,-179.808,7.948,149.457
C06368=1106.141,90.131,-58.062,-179.809,7.945,149.457
C06369=1106.146,89.882,-58.043,-179.811,7.941,149.457
C06370=1106.151,89.633,-58.024,-179.812,7.936,149.456
C06371=1106.156,89.384,-58.005,-179.813,7.933,149.455
C06372=1106.160,89.134,-57.986,-179.815,7.929,149.455
C06373=1106.165,88.886,-57.967,-179.816,7.925,149.454
C06374=1106.170,88.636,-57.949,-179.817,7.922,149.454
C06375=1106.174,88.387,-57.930,-179.818,7.918,149.454
C06376=1106.180,88.138,-57.911,-179.820,7.914,149.453
C06377=1106.184,87.888,-57.892,-179.821,7.911,149.452
C06378=1106.189,87.639,-57.873,-179.822,7.907,149.452
C06379=1106.194,87.390,-57.855,-179.823,7.903,149.451
C06380=1106.199,87.141,-57.835,-179.824,7.900,149.451
C06381=1106.203,86.891,-57.816,-179.825,7.895,149.450
C06382=1106.209,86.642,-57.798,-179.827,7.891,149.450
C06383=1106.213,86.393,-57.779,-179.828,7.888,149.449
C06384=1106.218,86.144,-57.761,-179.829,7.884,149.449
C06385=1106.223,85.895,-57.741,-179.831,7.880,149.448
C06386=1106.227,85.645,-57.723,-179.831,7.877,149.448
C06387=1106.233,85.396,-57.704,-179.833,7.873,149.447
C06388=1106.238,85.147,-57.686,-179.833,7.869,149.447
C06389=1106.242,84.897,-57.667,-179.835,7.865,149.446
C06390=1106.247,84.648,-57.648,-179.836,7.861,149.446
C06391=1106.252,84.399,-57.629,-179.837,7.858,149.445
C06392=1106.256,84.150,-57.611,-179.838,7.854,149.444
C06393=1106.261,83.901,-57.592,-179.839,7.851,149.444
C06394=1106.266,83.651,-57.573,-179.840,7.846,149.443
C06395=1106.270,83.402,-57.555,-179.842,7.842,149.443
C06396=1106.276,83.153,-57.536,-179.842,7.839,149.442
C06397=1106.280,82.903,-57.518,-179.844,7.835,149.442
C06398=1106.285,82.654,-57.499,-179.844,7.831,149.441
C06399=1106.291,82.405,-57.480,-179.846,7.828,149.441
C06400=1106.295,82.156,-57.461,-179.846,7.824,149.440
C06401=1106.300,81.906,-57.443,-179.848,7.820,149.440
C06402=1106.305,81.657,-57.425,-179.849,7.817,149.439
C06403=1106.309,81.408,-57.406,-179.850,7.813,149.439
C06404=1106.314,81.158,-57.388,-179.851,7.809,149.438
C06405=1106.319,80.909,-57.370,-179.852,7.805,149.437
C06406=1106.324,80.660,-57.350,-179.853,7.801,149.437
C06407=1106.329,80.411,-57.332,-179.854,7.798,149.436
C06408=1106.334,80.161,-57.314,-179.855,7.794,149.436
C06409=1106.339,79.913,-57.295,-179.856,7.791,149.435
C06410=1106.343,79.663,-57.277,-179.858,7.786,149.435
C06411=1106.348,79.413,-57.259,-179.859,7.783,149.434
C06412=1106.353,79.165,-57.240,-179.860,7.779,149.434
C06413=1106.357,78.915,-57.222,-179.861,7.776,149.433
C06414=1106.363,78.666,-57.203,-179.862,7.772,149.432
C06415=1106.367,78.452,-57.187,-179.863,7.768,149.432
C06416=1106.370,78.238,-57.172,-179.864,7.765,149.432
C06417=1106.375,78.025,-57.156,-179.864,7.762,149.431
C06418=1106.379,77.812,-57.140,-179.864,7.760,149.431
C06419=1106.383,77.598,-57.124,-179.865,7.756,149.430
C06420=1106.388,77.383,-57.109,-179.866,7.753,149.430
C06421=1106.391,77.169,-57.093,-179.867,7.750,149.429
C06422=1106.396,76.956,-57.077,-179.868,7.747,149.429
C06423=1106.401,76.707,-57.059,-179.869,7.743,149.428
C06424=1106.405,76.458,-57.041,-179.871,7.739,149.428
C06425=1106.410,76.208,-57.022,-179.872,7.735,149.427
C06426=1106.415,75.959,-57.004,-179.874,7.731,149.427
C06427=1106.420,75.710,-56.986,-179.875,7.727,149.426
C06428=1106.425,75.461,-56.968,-179.877,7.723,149.426
C06429=1106.429,75.211,-56.949,-179.878,7.719,149.425
C06430=1106.434,74.962,-56.931,-179.880,7.715,149.425
C06431=1106.439,74.712,-56.913,-179.881,7.711,149.424
C06432=1106.444,74.464,-56.895,-179.882,7.707,149.424
C06433=1106.449,74.215,-56.877,-179.883,7.703,149.423
C06434=1106.453,73.965,-56.858,-179.885,7.700,149.423
C06435=1106.458,73.716,-56.840,-179.886,7.696,149.422
C06436=1106.463,73.466,-56.823,-179.888,7.691,149.422
C06437=1106.468,73.217,-56.805,-179.889,7.687,149.421
C06438=1106.473,72.968,-56.786,-179.891,7.684,149.421
C06439=1106.478,72.719,-56.768,-179.892,7.679,149.420
C06440=1106.483,72.469,-56.750,-179.893,7.675,149.420
C06441=1106.488,72.219,-56.732,-179.894,7.672,149.419
C06442=1106.493,71.970,-56.714,-179.895,7.668,149.419
C06443=1106.497,71.721,-56.696,-179.897,7.664,149.418
C06444=1106.502,71.472,-56.678,-179.899,7.660,149.418
C06445=1106.507,71.223,-56.660,-179.900,7.656,149.417
C06446=1106.512,70.974,-56.642,-179.901,7.652,149.417
C06447=1106.516,70.724,-56.623,-179.903,7.648,149.416
C06448=1106.522,70.474,-56.606,-179.904,7.644,149.416
C06449=1106.527,70.225,-56.588,-179.905,7.641,149.415
C06450=1106.532,69.976,-56.570,-179.906,7.637,149.415
C06451=1106.536,69.726,-56.552,-179.908,7.632,149.414
C06452=1106.541,69.477,-56.534,-179.909,7.629,149.414
C06453=1106.546,69.228,-56.517,-179.911,7.625,149.413
C06454=1106.550,68.979,-56.499,-179.912,7.620,149.412
C06455=1106.555,68.730,-56.481,-179.913,7.616,149.412
C06456=1106.560,68.480,-56.463,-179.915,7.613,149.412
C06457=1106.565,68.230,-56.445,-179.915,7.609,149.411
C06458=1106.570,67.981,-56.427,-179.917,7.605,149.411
C06459=1106.575,67.732,-56.409,-179.918,7.601,149.410
C06460=1106.580,67.483,-56.391,-179.920,7.597,149.409
C06461=1106.585,67.233,-56.374,-179.921,7.593,149.409
C06462=1106.590,66.984,-56.356,-179.922,7.589,149.408
C06463=1106.594,66.735,-56.339,-179.923,7.586,149.408
C06464=1106.599,66.486,-56.321,-179.925,7.582,149.407
C06465=1106.604,66.236,-56.303,-179.926,7.578,149.407
C06466=1106.609,65.987,-56.285,-179.928,7.574,149.406
C06467=1106.614,65.738,-56.267,-179.929,7.569,149.406
C06468=1106.619,65.488,-56.250,-179.930,7.565,149.405
C06469=1106.624,65.239,-56.232,-179.932,7.562,149.405
C06470=1106.628,64.990,-56.215,-179.932,7.558,149.404
C06471=1106.633,64.776,-56.200,-179.934,7.554,149.404
C06472=1106.636,64.562,-56.184,-179.935,7.551,149.403
C06473=1106.641,64.348,-56.169,-179.936,7.548,149.403
C06474=1106.645,64.134,-56.154,-179.937,7.544,149.402
C06475=1106.649,63.921,-56.139,-179.938,7.541,149.402
C06476=1106.654,63.707,-56.124,-179.939,7.538,149.402
C06477=1106.657,63.493,-56.109,-179.940,7.535,149.401
C06478=1106.662,63.279,-56.094,-179.941,7.530,149.401
C06479=1106.667,63.029,-56.076,-179.942,7.527,149.400
C06480=1106.671,62.780,-56.059,-179.944,7.523,149.400
C06481=1106.676,62.531,-56.041,-179.945,7.519,149.399
C06482=1106.681,62.281,-56.024,-179.946,7.515,149.399
C06483=1106.686,62.032,-56.006,-179.948,7.511,149.398
C06484=1106.691,61.783,-55.989,-179.949,7.507,149.397
C06485=1106.695,61.534,-55.971,-179.950,7.503,149.397
C06486=1106.701,61.284,-55.954,-179.951,7.499,149.396
C06487=1106.705,61.035,-55.936,-179.952,7.495,149.396
C06488=1106.711,60.786,-55.920,-179.954,7.491,149.395
C06489=1106.716,60.537,-55.902,-179.955,7.487,149.395
C06490=1106.720,60.287,-55.885,-179.956,7.484,149.394
C06491=1106.725,60.038,-55.867,-179.957,7.480,149.394
C06492=1106.730,59.788,-55.850,-179.958,7.476,149.393
C06493=1106.734,59.539,-55.832,-179.960,7.471,149.392
C06494=1106.740,59.290,-55.815,-179.961,7.467,149.392
C06495=1106.745,59.040,-55.797,-179.962,7.464,149.391
C06496=1106.749,58.791,-55.780,-179.963,7.460,149.391
C06497=1106.754,58.541,-55.763,-179.964,7.456,149.390
C06498=1106.759,58.292,-55.745,-179.966,7.452,149.390
C06499=1106.764,58.043,-55.729,-179.967,7.448,149.389
C06500=1106.769,57.794,-55.711,-179.968,7.444,149.389
C06501=1106.774,57.544,-55.694,-179.969,7.440,149.388
C06502=1106.779,57.295,-55.677,-179.971,7.436,149.388
C06503=1106.784,57.046,-55.659,-179.972,7.432,149.387
C06504=1106.788,56.796,-55.642,-179.973,7.428,149.387
C06505=1106.793,56.546,-55.625,-179.974,7.425,149.386
C06506=1106.798,56.297,-55.608,-179.975,7.420,149.385
C06507=1106.803,56.048,-55.591,-179.976,7.416,149.385
C06508=1106.809,55.799,-55.573,-179.977,7.412,149.384
C06509=1106.813,55.550,-55.556,-179.979,7.408,149.384
C06510=1106.818,55.300,-55.539,-179.979,7.405,149.383
C06511=1106.823,55.050,-55.522,-179.981,7.401,149.383
C06512=1106.828,54.801,-55.505,-179.982,7.396,149.382
C06513=1106.832,54.552,-55.488,-179.983,7.392,149.381
C06514=1106.838,54.303,-55.471,-179.984,7.389,149.381
C06515=1106.842,54.053,-55.454,-179.985,7.385,149.380
C06516=1106.847,53.803,-55.437,-179.987,7.381,149.380
C06517=1106.852,53.554,-55.419,-179.988,7.376,149.379
C06518=1106.857,53.305,-55.402,-179.989,7.372,149.379
C06519=1106.862,53.056,-55.386,-179.990,7.369,149.378
C06520=1106.867,52.806,-55.368,-179.991,7.365,149.377
C06521=1106.872,52.557,-55.352,-179.993,7.361,149.377
C06522=1106.877,52.307,-55.334,-179.994,7.357,149.376
C06523=1106.882,52.059,-55.317,-179.994,7.353,149.376
C06524=1106.887,51.809,-55.300,-179.996,7.349,149.375
C06525=1106.891,51.559,-55.284,-179.997,7.345,149.375
C06526=1106.896,51.310,-55.266,-179.998,7.341,149.374
C06527=1106.900,51.096,-55.252,-179.999,7.337,149.374
C06528=1106.904,50.882,-55.237,-180.000,7.334,149.373
C06529=1106.908,50.668,-55.223,180.000,7.331,149.372
C06530=1106.913,50.454,-55.209,179.998,7.327,149.372
C06531=1106.917,50.240,-55.194,179.997,7.324,149.372
C06532=1106.921,50.026,-55.180,179.996,7.321,149.371
C06533=1106.925,49.813,-55.165,179.996,7.317,149.371
C06534=1106.930,49.599,-55.150,179.994,7.313,149.370
C06535=1106.935,49.350,-55.134,179.994,7.310,149.369
C06536=1106.940,49.100,-55.117,179.992,7.306,149.369
C06537=1106.945,48.851,-55.100,179.991,7.301,149.368
C06538=1106.949,48.601,-55.084,179.990,7.297,149.368
C06539=1106.955,48.352,-55.067,179.990,7.294,149.367
C06540=1106.960,48.103,-55.050,179.988,7.290,149.367
C06541=1106.964,47.853,-55.033,179.987,7.285,149.366
C06542=1106.969,47.604,-55.017,179.986,7.281,149.365
C06543=1106.975,47.355,-55.000,179.986,7.278,149.365
C06544=1106.979,47.105,-54.983,179.984,7.274,149.364
C06545=1106.984,46.856,-54.967,179.983,7.269,149.364
C06546=1106.989,46.607,-54.949,179.982,7.265,149.363
C06547=1106.994,46.357,-54.933,179.981,7.262,149.362
C06548=1106.999,46.108,-54.917,179.980,7.258,149.362
C06549=1107.004,45.858,-54.901,179.979,7.253,149.361
C06550=1107.009,45.608,-54.883,179.978,7.249,149.360
C06551=1107.014,45.360,-54.867,179.977,7.246,149.360
C06552=1107.018,45.110,-54.850,179.976,7.241,149.359
C06553=1107.023,44.861,-54.834,179.975,7.237,149.359
C06554=1107.029,44.611,-54.817,179.974,7.233,149.358
C06555=1107.033,44.362,-54.800,179.973,7.230,149.357
C06556=1107.038,44.112,-54.784,179.972,7.225,149.357
C06557=1107.043,43.863,-54.768,179.971,7.221,149.356
C06558=1107.048,43.613,-54.751,179.969,7.217,149.356
C06559=1107.053,43.364,-54.734,179.969,7.214,149.355
C06560=1107.058,43.115,-54.718,179.968,7.209,149.354
C06561=1107.063,42.865,-54.702,179.967,7.205,149.354
C06562=1107.068,42.616,-54.685,179.966,7.201,149.353
C06563=1107.073,42.366,-54.668,179.965,7.197,149.352
C06564=1107.077,42.117,-54.651,179.964,7.193,149.352
C06565=1107.083,41.867,-54.636,179.963,7.189,149.351
C06566=1107.087,41.618,-54.619,179.962,7.185,149.351
C06567=1107.092,41.369,-54.603,179.961,7.181,149.350
C06568=1107.097,41.120,-54.586,179.960,7.177,149.349
C06569=1107.103,40.870,-54.570,179.959,7.172,149.349
C06570=1107.107,40.621,-54.553,179.958,7.168,149.348
C06571=1107.112,40.371,-54.537,179.957,7.165,149.347
C06572=1107.117,40.122,-54.521,179.956,7.160,149.347
C06573=1107.122,39.872,-54.504,179.955,7.156,149.346
C06574=1107.127,39.623,-54.488,179.955,7.153,149.345
C06575=1107.132,39.373,-54.472,179.954,7.148,149.345
C06576=1107.137,39.124,-54.455,179.953,7.144,149.344
C06577=1107.142,38.875,-54.439,179.951,7.140,149.344
C06578=1107.147,38.625,-54.423,179.951,7.136,149.343
C06579=1107.152,38.376,-54.406,179.950,7.132,149.342
C06580=1107.157,38.126,-54.391,179.949,7.128,149.342
C06581=1107.162,37.877,-54.374,179.947,7.124,149.341
C06582=1107.167,37.628,-54.358,179.947,7.120,149.340
C06583=1107.171,37.414,-54.344,179.946,7.116,149.340
C06584=1107.175,37.200,-54.330,179.945,7.113,149.339
C06585=1107.179,36.986,-54.316,179.945,7.109,149.339
C06586=1107.184,36.771,-54.302,179.944,7.106,149.338
C06587=1107.188,36.558,-54.288,179.943,7.102,149.338
C06588=1107.193,36.344,-54.274,179.942,7.098,149.337
C06589=1107.197,36.130,-54.261,179.941,7.095,149.336
C06590=1107.201,35.916,-54.246,179.941,7.092,149.336
C06591=1107.206,35.666,-54.230,179.940,7.087,149.335
C06592=1107.211,35.417,-54.214,179.939,7.084,149.334
C06593=1107.215,35.167,-54.198,179.938,7.079,149.334
C06594=1107.221,34.918,-54.183,179.937,7.075,149.333
C06595=1107.226,34.669,-54.166,179.936,7.071,149.333
C06596=1107.231,34.419,-54.150,179.936,7.067,149.332
C06597=1107.236,34.170,-54.134,179.935,7.063,149.331
C06598=1107.241,33.920,-54.118,179.934,7.058,149.330
C06599=1107.246,33.671,-54.102,179.933,7.054,149.330
C06600=1107.250,33.421,-54.086,179.932,7.050,149.329
C06601=1107.255,33.173,-54.070,179.931,7.046,149.328
C06602=1107.260,32.923,-54.054,179.930,7.042,149.328
C06603=1107.265,32.673,-54.038,179.930,7.038,149.327
C06604=1107.270,32.424,-54.022,179.929,7.034,149.326
C06605=1107.275,32.174,-54.006,179.928,7.030,149.326
C06606=1107.280,31.925,-53.991,179.927,7.025,149.325
C06607=1107.285,31.675,-53.974,179.927,7.021,149.324
C06608=1107.290,31.426,-53.958,179.926,7.017,149.324
C06609=1107.295,31.177,-53.943,179.925,7.013,149.323
C06610=1107.300,30.927,-53.926,179.924,7.009,149.322
C06611=1107.305,30.678,-53.911,179.923,7.005,149.322
C06612=1107.309,30.428,-53.895,179.923,7.000,149.321
C06613=1107.314,30.179,-53.879,179.921,6.996,149.320
C06614=1107.320,29.930,-53.863,179.921,6.992,149.319
C06615=1107.325,29.680,-53.847,179.920,6.988,149.319
C06616=1107.330,29.431,-53.831,179.919,6.983,149.318
C06617=1107.334,29.181,-53.815,179.918,6.979,149.317
C06618=1107.339,28.932,-53.800,179.918,6.976,149.317
C06619=1107.345,28.682,-53.784,179.917,6.971,149.316
C06620=1107.349,28.432,-53.769,179.916,6.967,149.315
C06621=1107.354,28.183,-53.752,179.915,6.962,149.314
C06622=1107.360,27.934,-53.737,179.915,6.959,149.314
C06623=1107.364,27.684,-53.721,179.914,6.955,149.313
C06624=1107.369,27.435,-53.706,179.913,6.950,149.312
C06625=1107.375,27.185,-53.690,179.913,6.946,149.311
C06626=1107.379,26.936,-53.673,179.912,6.942,149.311
C06627=1107.384,26.686,-53.658,179.911,6.937,149.310
C06628=1107.389,26.437,-53.643,179.910,6.933,149.309
C06629=1107.394,26.187,-53.627,179.910,6.929,149.309
C06630=1107.399,25.938,-53.611,179.909,6.925,149.308
C06631=1107.405,25.688,-53.596,179.908,6.920,149.307
C06632=1107.409,25.439,-53.580,179.907,6.916,149.306
C06633=1107.414,25.190,-53.564,179.907,6.912,149.306
C06634=1107.419,24.940,-53.548,179.906,6.908,149.305
C06635=1107.425,24.691,-53.533,179.905,6.904,149.304
C06636=1107.429,24.441,-53.518,179.905,6.900,149.303
C06637=1107.434,24.192,-53.502,179.904,6.895,149.303
C06638=1107.439,23.942,-53.486,179.903,6.891,149.302
C06639=1107.443,23.728,-53.473,179.902,6.888,149.301
C06640=1107.447,23.514,-53.460,179.902,6.884,149.301
C06641=1107.452,23.300,-53.446,179.901,6.880,149.300
C06642=1107.456,23.086,-53.433,179.900,6.876,149.299
C06643=1107.460,22.872,-53.420,179.900,6.873,149.299
C06644=1107.465,22.658,-53.407,179.900,6.869,149.298
C06645=1107.469,22.444,-53.394,179.899,6.866,149.297
C06646=1107.473,22.230,-53.380,179.898,6.861,149.297
C06647=1107.478,21.980,-53.364,179.898,6.857,149.296
C06648=1107.483,21.731,-53.349,179.897,6.853,149.295
C06649=1107.488,21.482,-53.334,179.896,6.848,149.294
C06650=1107.493,21.232,-53.318,179.896,6.845,149.294
C06651=1107.498,20.982,-53.303,179.895,6.840,149.293
C06652=1107.503,20.733,-53.287,179.894,6.836,149.292
C06653=1107.508,20.484,-53.272,179.894,6.831,149.291
C06654=1107.513,20.235,-53.257,179.893,6.828,149.291
C06655=1107.518,19.984,-53.241,179.893,6.823,149.290
C06656=1107.523,19.735,-53.226,179.892,6.819,149.289
C06657=1107.528,19.485,-53.211,179.891,6.814,149.288
C06658=1107.533,19.236,-53.196,179.891,6.810,149.288
C06659=1107.538,18.987,-53.180,179.890,6.806,149.287
C06660=1107.543,18.737,-53.165,179.889,6.801,149.286
C06661=1107.548,18.488,-53.149,179.889,6.797,149.285
C06662=1107.553,18.238,-53.134,179.889,6.793,149.284
C06663=1107.558,17.989,-53.119,179.888,6.788,149.284
C06664=1107.564,17.739,-53.104,179.887,6.784,149.283
C06665=1107.568,17.489,-53.088,179.887,6.779,149.282
C06666=1107.573,17.240,-53.073,179.886,6.776,149.281
C06667=1107.578,16.991,-53.058,179.886,6.771,149.280
C06668=1107.583,16.741,-53.042,179.885,6.766,149.280
C06669=1107.588,16.492,-53.028,179.884,6.762,149.279
C06670=1107.593,16.242,-53.012,179.884,6.758,149.278
C06671=1107.598,15.993,-52.997,179.883,6.754,149.277
C06672=1107.603,15.743,-52.982,179.882,6.749,149.276
C06673=1107.608,15.494,-52.967,179.882,6.745,149.275
C06674=1107.613,15.244,-52.952,179.882,6.740,149.275
C06675=1107.618,14.995,-52.937,179.881,6.736,149.274
C06676=1107.623,14.746,-52.921,179.880,6.731,149.273
C06677=1107.628,14.496,-52.907,179.880,6.727,149.272
C06678=1107.634,14.246,-52.891,179.879,6.723,149.271
C06679=1107.638,13.997,-52.876,179.879,6.718,149.271
C06680=1107.642,13.748,-52.861,179.878,6.714,149.270
C06681=1107.648,13.498,-52.846,179.878,6.710,149.269
C06682=1107.653,13.248,-52.831,179.878,6.705,149.268
C06683=1107.658,12.999,-52.815,179.877,6.701,149.267
C06684=1107.663,12.749,-52.801,179.876,6.696,149.266
C06685=1107.668,12.500,-52.786,179.876,6.691,149.265
C06686=1107.673,12.250,-52.771,179.876,6.687,149.265
C06687=1107.678,12.001,-52.756,179.875,6.683,149.264
C06688=1107.683,11.752,-52.741,179.874,6.678,149.263
C06689=1107.688,11.502,-52.726,179.874,6.674,149.262
C06690=1107.693,11.253,-52.711,179.874,6.670,149.261
C06691=1107.699,11.003,-52.697,179.873,6.665,149.260
C06692=1107.703,10.754,-52.682,179.872,6.660,149.259
C06693=1107.708,10.504,-52.666,179.872,6.656,149.259
C06694=1107.713,10.254,-52.651,179.872,6.652,149.258
C06695=1107.717,10.041,-52.639,179.871,6.647,149.257
C06696=1107.722,9.826,-52.626,179.871,6.644,149.256
C06697=1107.726,9.612,-52.613,179.871,6.640,149.255
C06698=1107.730,9.398,-52.600,179.870,6.636,149.255
C06699=1107.735,9.184,-52.588,179.870,6.632,149.254
C06700=1107.739,8.970,-52.575,179.869,6.628,149.253
C06701=1107.744,8.755,-52.562,179.869,6.625,149.253
C06702=1107.747,8.541,-52.549,179.869,6.621,149.252
C06703=1107.752,8.292,-52.535,179.868,6.616,149.251
C06704=1107.758,8.042,-52.519,179.867,6.612,149.250
C06705=1107.763,7.792,-52.505,179.867,6.607,149.249
C06706=1107.768,7.543,-52.491,179.866,6.602,149.248
C06707=1107.772,7.294,-52.476,179.866,6.598,149.247
C06708=1107.778,7.044,-52.461,179.865,6.593,149.247
C06709=1107.783,6.795,-52.446,179.864,6.588,149.246
C06710=1107.788,6.545,-52.431,179.864,6.584,149.245
C06711=1107.792,6.296,-52.416,179.863,6.579,149.244
C06712=1107.798,6.046,-52.402,179.863,6.574,149.243
C06713=1107.803,5.796,-52.387,179.861,6.570,149.243
C06714=1107.808,5.547,-52.372,179.861,6.565,149.242
C06715=1107.813,5.298,-52.358,179.860,6.561,149.241
C06716=1107.818,5.049,-52.343,179.860,6.556,149.240
C06717=1107.823,4.799,-52.328,179.859,6.552,149.239
C06718=1107.828,4.549,-52.314,179.858,6.547,149.238
C06719=1107.833,4.300,-52.299,179.858,6.542,149.238
C06720=1107.838,4.050,-52.285,179.857,6.537,149.237
C06721=1107.844,3.800,-52.270,179.856,6.533,149.236
C06722=1107.848,3.551,-52.255,179.856,6.528,149.235
C06723=1107.853,3.301,-52.241,179.855,6.524,149.234
C06724=1107.858,3.052,-52.227,179.855,6.519,149.233
C06725=1107.863,2.802,-52.212,179.854,6.515,149.233
C06726=1107.868,2.553,-52.197,179.853,6.510,149.232
C06727=1107.873,2.303,-52.183,179.853,6.505,149.231
C06728=1107.878,2.053,-52.168,179.853,6.501,149.230
C06729=1107.884,1.804,-52.154,179.852,6.497,149.229
C06730=1107.889,1.555,-52.139,179.851,6.492,149.228
C06731=1107.894,1.305,-52.125,179.851,6.488,149.228
C06732=1107.899,1.056,-52.111,179.850,6.483,149.227
C06733=1107.904,0.806,-52.096,179.849,6.479,149.226
C06734=1107.908,0.556,-52.082,179.849,6.474,149.225
C06735=1107.913,0.307,-52.067,179.848,6.469,149.224
C06736=1107.918,0.057,-52.053,179.847,6.465,149.224
C06737=1107.924,-0.192,-52.039,179.846,6.460,149.223
C06738=1107.929,-0.442,-52.024,179.846,6.455,149.222
C06739=1107.934,-0.691,-52.010,179.845,6.451,149.221
C06740=1107.939,-0.941,-51.995,179.844,6.446,149.220
C06741=1107.944,-1.190,-51.980,179.844,6.442,149.219
C06742=1107.949,-1.440,-51.966,179.844,6.438,149.218
C06743=1107.954,-1.689,-51.952,179.843,6.433,149.218
C06744=1107.959,-1.938,-51.938,179.842,6.429,149.217
C06745=1107.964,-2.188,-51.924,179.842,6.424,149.216
C06746=1107.969,-2.438,-51.909,179.841,6.420,149.215
C06747=1107.974,-2.688,-51.895,179.840,6.415,149.214
C06748=1107.979,-2.937,-51.881,179.840,6.410,149.213
C06749=1107.985,-3.186,-51.867,179.839,6.405,149.213
C06750=1107.990,-3.436,-51.853,179.838,6.401,149.212
C06751=1107.994,-3.651,-51.840,179.838,6.398,149.211
C06752=1107.998,-3.865,-51.828,179.838,6.394,149.210
C06753=1108.002,-4.079,-51.816,179.837,6.389,149.210
C06754=1108.006,-4.293,-51.804,179.837,6.386,149.209
C06755=1108.011,-4.507,-51.792,179.836,6.382,149.208
C06756=1108.015,-4.721,-51.780,179.835,6.378,149.208
C06757=1108.019,-4.936,-51.767,179.835,6.374,149.207
C06758=1108.024,-5.150,-51.755,179.835,6.370,149.206
C06759=1108.029,-5.399,-51.741,179.834,6.366,149.205
C06760=1108.034,-5.648,-51.727,179.833,6.361,149.205
C06761=1108.039,-5.898,-51.713,179.833,6.357,149.204
C06762=1108.044,-6.148,-51.699,179.832,6.352,149.203
C06763=1108.049,-6.398,-51.685,179.831,6.348,149.202
C06764=1108.055,-6.647,-51.671,179.831,6.343,149.201
C06765=1108.060,-6.897,-51.657,179.831,6.339,149.200
C06766=1108.065,-7.146,-51.643,179.831,6.334,149.199
C06767=1108.070,-7.396,-51.628,179.830,6.330,149.199
C06768=1108.075,-7.645,-51.614,179.829,6.325,149.198
C06769=1108.079,-7.895,-51.601,179.828,6.320,149.197
C06770=1108.084,-8.144,-51.586,179.828,6.316,149.196
C06771=1108.089,-8.394,-51.572,179.827,6.311,149.195
C06772=1108.095,-8.644,-51.559,179.826,6.307,149.195
C06773=1108.100,-8.893,-51.545,179.827,6.303,149.194
C06774=1108.105,-9.143,-51.530,179.826,6.298,149.193
C06775=1108.111,-9.392,-51.517,179.825,6.294,149.192
C06776=1108.115,-9.641,-51.503,179.825,6.289,149.191
C06777=1108.120,-9.892,-51.489,179.824,6.284,149.190
C06778=1108.126,-10.141,-51.475,179.824,6.280,149.189
C06779=1108.131,-10.391,-51.461,179.823,6.275,149.189
C06780=1108.136,-10.640,-51.447,179.822,6.271,149.188
C06781=1108.140,-10.890,-51.433,179.822,6.267,149.187
C06782=1108.146,-11.139,-51.420,179.822,6.262,149.186
C06783=1108.151,-11.389,-51.406,179.821,6.258,149.185
C06784=1108.156,-11.639,-51.391,179.820,6.253,149.184
C06785=1108.160,-11.887,-51.378,179.820,6.248,149.184
C06786=1108.166,-12.138,-51.365,179.819,6.243,149.183
C06787=1108.171,-12.387,-51.350,179.819,6.239,149.182
C06788=1108.176,-12.636,-51.336,179.818,6.234,149.181
C06789=1108.181,-12.886,-51.323,179.818,6.230,149.180
C06790=1108.186,-13.135,-51.309,179.817,6.226,149.179
C06791=1108.191,-13.385,-51.295,179.817,6.221,149.178
C06792=1108.197,-13.636,-51.282,179.816,6.216,149.177
C06793=1108.201,-13.884,-51.268,179.815,6.212,149.177
C06794=1108.206,-14.134,-51.254,179.815,6.207,149.176
C06795=1108.212,-14.384,-51.240,179.814,6.202,149.175
C06796=1108.216,-14.633,-51.227,179.814,6.199,149.174
C06797=1108.222,-14.883,-51.214,179.814,6.194,149.173
C06798=1108.227,-15.132,-51.200,179.813,6.189,149.172
C06799=1108.231,-15.382,-51.186,179.813,6.184,149.171
C06800=1108.237,-15.632,-51.172,179.812,6.180,149.171
C06801=1108.242,-15.881,-51.158,179.811,6.175,149.170
C06802=1108.247,-16.131,-51.146,179.811,6.171,149.169
C06803=1108.252,-16.380,-51.132,179.810,6.166,149.168
C06804=1108.258,-16.630,-51.118,179.811,6.162,149.167
C06805=1108.262,-16.879,-51.105,179.810,6.157,149.166
C06806=1108.267,-17.129,-51.090,179.810,6.152,149.165
C06807=1108.272,-17.343,-51.079,179.809,6.148,149.165
C06808=1108.277,-17.557,-51.067,179.808,6.145,149.164
C06809=1108.280,-17.772,-51.056,179.808,6.141,149.163
C06810=1108.284,-17.986,-51.044,179.807,6.136,149.162
C06811=1108.289,-18.201,-51.033,179.807,6.133,149.162
C06812=1108.294,-18.415,-51.021,179.807,6.129,149.161
C06813=1108.298,-18.629,-51.009,179.806,6.125,149.160
C06814=1108.302,-18.843,-50.999,179.806,6.121,149.159
C06815=1108.307,-19.093,-50.984,179.806,6.116,149.158
C06816=1108.313,-19.342,-50.972,179.805,6.111,149.158
C06817=1108.318,-19.592,-50.957,179.805,6.106,149.157
C06818=1108.323,-19.842,-50.944,179.805,6.102,149.156
C06819=1108.328,-20.091,-50.931,179.804,6.098,149.155
C06820=1108.333,-20.341,-50.917,179.804,6.093,149.154
C06821=1108.338,-20.591,-50.904,179.803,6.089,149.153
C06822=1108.344,-20.840,-50.891,179.803,6.084,149.152
C06823=1108.348,-21.090,-50.878,179.802,6.079,149.151
C06824=1108.354,-21.339,-50.864,179.802,6.074,149.150
C06825=1108.358,-21.589,-50.851,179.802,6.069,149.149
C06826=1108.364,-21.839,-50.837,179.801,6.065,149.148
C06827=1108.368,-22.088,-50.824,179.801,6.061,149.148
C06828=1108.374,-22.338,-50.811,179.801,6.056,149.147
C06829=1108.379,-22.588,-50.798,179.800,6.051,149.146
C06830=1108.384,-22.837,-50.784,179.800,6.047,149.145
C06831=1108.389,-23.087,-50.771,179.799,6.042,149.144
C06832=1108.395,-23.336,-50.758,179.799,6.037,149.143
C06833=1108.399,-23.586,-50.745,179.798,6.032,149.142
C06834=1108.405,-23.835,-50.731,179.798,6.028,149.141
C06835=1108.410,-24.085,-50.718,179.797,6.023,149.140
C06836=1108.415,-24.335,-50.705,179.797,6.018,149.139
C06837=1108.420,-24.584,-50.691,179.797,6.013,149.138
C06838=1108.425,-24.834,-50.678,179.796,6.008,149.137
C06839=1108.430,-25.083,-50.665,179.797,6.004,149.137
C06840=1108.435,-25.333,-50.652,179.796,6.000,149.136
C06841=1108.441,-25.583,-50.639,179.796,5.995,149.135
C06842=1108.445,-25.832,-50.626,179.796,5.990,149.134
C06843=1108.451,-26.082,-50.612,179.796,5.986,149.133
C06844=1108.456,-26.331,-50.599,179.795,5.981,149.132
C06845=1108.460,-26.581,-50.586,179.795,5.976,149.131
C06846=1108.466,-26.831,-50.573,179.795,5.972,149.130
C06847=1108.471,-27.080,-50.560,179.795,5.967,149.129
C06848=1108.476,-27.330,-50.547,179.796,5.963,149.128
C06849=1108.481,-27.579,-50.534,179.795,5.958,149.127
C06850=1108.486,-27.829,-50.521,179.795,5.954,149.126
C06851=1108.492,-28.079,-50.508,179.795,5.950,149.125
C06852=1108.497,-28.328,-50.495,179.795,5.945,149.124
C06853=1108.501,-28.578,-50.482,179.795,5.941,149.123
C06854=1108.507,-28.827,-50.468,179.795,5.937,149.122
C06855=1108.512,-29.077,-50.456,179.795,5.932,149.121
C06856=1108.517,-29.327,-50.443,179.795,5.928,149.120
C06857=1108.522,-29.576,-50.429,179.794,5.923,149.119
C06858=1108.527,-29.826,-50.416,179.794,5.919,149.118
C06859=1108.532,-30.076,-50.404,179.794,5.915,149.118
C06860=1108.537,-30.325,-50.391,179.794,5.910,149.117
C06861=1108.543,-30.575,-50.378,179.794,5.906,149.116
C06862=1108.548,-30.824,-50.365,179.793,5.901,149.115
C06863=1108.552,-31.039,-50.354,179.793,5.897,149.114
C06864=1108.556,-31.253,-50.343,179.793,5.894,149.113
C06865=1108.561,-31.468,-50.332,179.793,5.890,149.112
C06866=1108.565,-31.682,-50.321,179.793,5.886,149.112
C06867=1108.570,-31.897,-50.310,179.792,5.882,149.111
C06868=1108.574,-32.110,-50.298,179.792,5.878,149.110
C06869=1108.579,-32.325,-50.287,179.792,5.874,149.109
C06870=1108.583,-32.539,-50.276,179.791,5.871,149.109
C06871=1108.588,-32.789,-50.263,179.791,5.866,149.108
C06872=1108.593,-33.039,-50.250,179.791,5.862,149.107
C06873=1108.598,-33.289,-50.238,179.791,5.857,149.106
C06874=1108.603,-33.538,-50.226,179.790,5.853,149.105
C06875=1108.608,-33.788,-50.213,179.790,5.849,149.104
C06876=1108.614,-34.038,-50.199,179.790,5.844,149.103
C06877=1108.619,-34.287,-50.187,179.789,5.839,149.102
C06878=1108.624,-34.537,-50.174,179.789,5.835,149.101
C06879=1108.629,-34.786,-50.161,179.789,5.831,149.101
C06880=1108.634,-35.036,-50.149,179.788,5.826,149.100
C06881=1108.640,-35.285,-50.135,179.788,5.822,149.099
C06882=1108.644,-35.535,-50.122,179.787,5.817,149.098
C06883=1108.649,-35.785,-50.110,179.787,5.813,149.097
C06884=1108.654,-36.034,-50.097,179.787,5.808,149.096
C06885=1108.660,-36.284,-50.085,179.786,5.803,149.095
C06886=1108.665,-36.534,-50.072,179.786,5.799,149.095
C06887=1108.670,-36.783,-50.059,179.785,5.794,149.094
C06888=1108.675,-37.033,-50.047,179.785,5.790,149.093
C06889=1108.680,-37.282,-50.034,179.784,5.785,149.092
C06890=1108.686,-37.531,-50.021,179.784,5.780,149.091
C06891=1108.690,-37.782,-50.009,179.783,5.775,149.090
C06892=1108.696,-38.031,-49.997,179.783,5.771,149.089
C06893=1108.701,-38.281,-49.984,179.783,5.767,149.088
C06894=1108.707,-38.530,-49.971,179.783,5.762,149.087
C06895=1108.711,-38.780,-49.958,179.782,5.757,149.086
C06896=1108.716,-39.030,-49.946,179.781,5.753,149.086
C06897=1108.722,-39.280,-49.933,179.781,5.748,149.085
C06898=1108.727,-39.529,-49.921,179.780,5.743,149.084
C06899=1108.732,-39.778,-49.908,179.779,5.738,149.083
C06900=1108.737,-40.028,-49.896,179.779,5.733,149.082
C06901=1108.742,-40.278,-49.883,179.778,5.728,149.081
C06902=1108.747,-40.527,-49.871,179.778,5.723,149.080
C06903=1108.752,-40.777,-49.859,179.778,5.719,149.079
C06904=1108.757,-41.027,-49.846,179.778,5.714,149.078
C06905=1108.763,-41.276,-49.834,179.777,5.709,149.077
C06906=1108.768,-41.526,-49.822,179.776,5.704,149.076
C06907=1108.773,-41.776,-49.809,179.776,5.699,149.075
C06908=1108.778,-42.025,-49.796,179.775,5.694,149.075
C06909=1108.783,-42.275,-49.784,179.775,5.689,149.074
C06910=1108.788,-42.525,-49.772,179.774,5.683,149.072
C06911=1108.793,-42.774,-49.759,179.774,5.679,149.072
C06912=1108.799,-43.024,-49.747,179.773,5.674,149.071
C06913=1108.804,-43.273,-49.734,179.774,5.670,149.070
C06914=1108.809,-43.523,-49.723,179.774,5.664,149.068
C06915=1108.814,-43.773,-49.710,179.774,5.659,149.067
C06916=1108.819,-44.022,-49.697,179.774,5.655,149.066
C06917=1108.824,-44.272,-49.685,179.774,5.650,149.065
C06918=1108.830,-44.522,-49.673,179.774,5.645,149.064
C06919=1108.834,-44.737,-49.663,179.775,5.641,149.063
C06920=1108.839,-44.951,-49.651,179.775,5.637,149.062
C06921=1108.843,-45.165,-49.641,179.775,5.633,149.061
C06922=1108.848,-45.379,-49.631,179.775,5.629,149.060
C06923=1108.852,-45.594,-49.620,179.775,5.625,149.059
C06924=1108.857,-45.809,-49.610,179.775,5.621,149.059
C06925=1108.861,-46.023,-49.599,179.776,5.618,149.058
C06926=1108.865,-46.238,-49.589,179.776,5.614,149.057
C06927=1108.870,-46.487,-49.576,179.776,5.608,149.056
C06928=1108.876,-46.737,-49.564,179.776,5.603,149.054
C06929=1108.881,-46.987,-49.552,179.777,5.599,149.053
C06930=1108.886,-47.236,-49.540,179.776,5.594,149.052
C06931=1108.891,-47.486,-49.527,179.776,5.589,149.051
C06932=1108.896,-47.735,-49.516,179.777,5.585,149.050
C06933=1108.901,-47.985,-49.503,179.776,5.580,149.049
C06934=1108.907,-48.235,-49.491,179.777,5.576,149.048
C06935=1108.912,-48.484,-49.479,179.777,5.571,149.047
C06936=1108.917,-48.734,-49.467,179.777,5.566,149.046
C06937=1108.923,-48.984,-49.455,179.777,5.562,149.045
C06938=1108.928,-49.233,-49.443,179.778,5.556,149.044
C06939=1108.932,-49.484,-49.431,179.778,5.551,149.042
C06940=1108.937,-49.733,-49.418,179.778,5.547,149.042
C06941=1108.942,-49.983,-49.406,179.778,5.542,149.040
C06942=1108.947,-50.232,-49.394,179.779,5.538,149.039
C06943=1108.953,-50.482,-49.382,179.778,5.533,149.038
C06944=1108.958,-50.732,-49.370,179.778,5.528,149.037
C06945=1108.963,-50.981,-49.358,179.779,5.524,149.036
C06946=1108.968,-51.231,-49.346,179.778,5.519,149.035
C06947=1108.974,-51.481,-49.334,179.779,5.514,149.034
C06948=1108.979,-51.730,-49.322,179.779,5.510,149.033
C06949=1108.984,-51.980,-49.310,179.779,5.505,149.032
C06950=1108.989,-52.230,-49.298,179.779,5.500,149.031
C06951=1108.994,-52.479,-49.286,179.780,5.495,149.030
C06952=1108.999,-52.729,-49.274,179.779,5.491,149.029
C06953=1109.005,-52.979,-49.262,179.780,5.486,149.027
C06954=1109.009,-53.228,-49.250,179.780,5.481,149.026
C06955=1109.015,-53.478,-49.238,179.780,5.476,149.025
C06956=1109.021,-53.727,-49.227,179.780,5.472,149.024
C06957=1109.026,-53.977,-49.215,179.780,5.467,149.023
C06958=1109.030,-54.226,-49.203,179.780,5.462,149.022
C06959=1109.036,-54.476,-49.191,179.781,5.458,149.021
C06960=1109.041,-54.726,-49.179,179.781,5.453,149.020
C06961=1109.047,-54.976,-49.167,179.780,5.448,149.019
C06962=1109.051,-55.225,-49.155,179.781,5.444,149.018
C06963=1109.057,-55.475,-49.143,179.781,5.438,149.017
C06964=1109.062,-55.725,-49.131,179.781,5.435,149.016
C06965=1109.067,-55.974,-49.120,179.781,5.429,149.015
C06966=1109.072,-56.224,-49.107,179.781,5.425,149.014
C06967=1109.077,-56.474,-49.096,179.782,5.420,149.012
C06968=1109.082,-56.723,-49.084,179.782,5.415,149.011
C06969=1109.087,-56.973,-49.072,179.781,5.410,149.010
C06970=1109.093,-57.223,-49.061,179.782,5.406,149.009
C06971=1109.097,-57.473,-49.049,179.782,5.401,149.008
C06972=1109.103,-57.722,-49.037,179.782,5.396,149.007
C06973=1109.108,-57.972,-49.025,179.782,5.392,149.006
C06974=1109.113,-58.221,-49.014,179.782,5.387,149.005
C06975=1109.118,-58.436,-49.004,179.782,5.383,149.004
C06976=1109.122,-58.651,-48.994,179.782,5.379,149.003
C06977=1109.126,-58.865,-48.983,179.783,5.375,149.002
C06978=1109.131,-59.079,-48.973,179.783,5.371,149.001
C06979=1109.135,-59.294,-48.963,179.782,5.367,149.000
C06980=1109.140,-59.509,-48.953,179.783,5.363,149.000
C06981=1109.144,-59.724,-48.943,179.783,5.359,148.999
C06982=1109.149,-59.938,-48.934,179.783,5.355,148.998
C06983=1109.154,-60.187,-48.921,179.783,5.350,148.997
C06984=1109.159,-60.437,-48.909,179.782,5.345,148.996
C06985=1109.164,-60.687,-48.898,179.782,5.340,148.995
C06986=1109.170,-60.937,-48.886,179.781,5.335,148.994
C06987=1109.174,-61.186,-48.875,179.781,5.330,148.993
C06988=1109.180,-61.436,-48.863,179.781,5.325,148.992
C06989=1109.185,-61.685,-48.852,179.781,5.320,148.991
C06990=1109.190,-61.935,-48.840,179.780,5.315,148.990
C06991=1109.195,-62.185,-48.829,179.780,5.310,148.989
C06992=1109.201,-62.435,-48.817,179.779,5.305,148.988
C06993=1109.206,-62.685,-48.805,179.779,5.300,148.987
C06994=1109.211,-62.934,-48.794,179.779,5.295,148.986
C06995=1109.217,-63.183,-48.782,179.779,5.290,148.985
C06996=1109.221,-63.433,-48.771,179.779,5.285,148.984
C06997=1109.227,-63.683,-48.759,179.778,5.280,148.983
C06998=1109.231,-63.933,-48.748,179.777,5.274,148.982
C06999=1109.237,-64.183,-48.736,179.778,5.269,148.981
C07000=1109.243,-64.432,-48.726,179.777,5.265,148.980
C07001=1109.248,-64.682,-48.714,179.777,5.259,148.978
C07002=1109.253,-64.932,-48.703,179.777,5.255,148.978
C07003=1109.257,-65.181,-48.691,179.777,5.250,148.976
C07004=1109.263,-65.431,-48.679,179.777,5.245,148.975
C07005=1109.268,-65.680,-48.668,179.776,5.239,148.974
C07006=1109.273,-65.930,-48.657,179.776,5.234,148.973
C07007=1109.278,-66.180,-48.645,179.776,5.229,148.972
C07008=1109.284,-66.430,-48.633,179.776,5.224,148.971
C07009=1109.289,-66.679,-48.623,179.776,5.219,148.970
C07010=1109.295,-66.929,-48.611,179.776,5.214,148.969
C07011=1109.299,-67.179,-48.600,179.776,5.209,148.968
C07012=1109.304,-67.428,-48.589,179.775,5.203,148.967
C07013=1109.310,-67.678,-48.577,179.775,5.198,148.966
C07014=1109.315,-67.928,-48.567,179.775,5.193,148.965
C07015=1109.320,-68.178,-48.555,179.775,5.188,148.964
C07016=1109.325,-68.427,-48.543,179.775,5.183,148.962
C07017=1109.330,-68.676,-48.533,179.775,5.178,148.961
C07018=1109.336,-68.927,-48.521,179.775,5.173,148.960
C07019=1109.341,-69.176,-48.510,179.775,5.168,148.959
C07020=1109.346,-69.425,-48.499,179.774,5.162,148.958
C07021=1109.352,-69.675,-48.487,179.775,5.157,148.957
C07022=1109.357,-69.926,-48.477,179.774,5.152,148.956
C07023=1109.363,-70.175,-48.465,179.774,5.147,148.955
C07024=1109.367,-70.424,-48.454,179.774,5.142,148.954
C07025=1109.372,-70.674,-48.443,179.775,5.137,148.952
C07026=1109.377,-70.924,-48.432,179.774,5.132,148.951
C07027=1109.383,-71.174,-48.420,179.774,5.127,148.950
C07028=1109.388,-71.423,-48.409,179.774,5.122,148.949
C07029=1109.393,-71.673,-48.399,179.775,5.117,148.948
C07030=1109.399,-71.923,-48.387,179.775,5.111,148.947
C07031=1109.402,-72.137,-48.378,179.774,5.107,148.946
C07032=1109.408,-72.352,-48.369,179.774,5.102,148.945
C07033=1109.412,-72.567,-48.359,179.774,5.098,148.944
C07034=1109.417,-72.781,-48.349,179.774,5.093,148.943
C07035=1109.420,-72.996,-48.340,179.775,5.089,148.942
C07036=1109.425,-73.211,-48.330,179.774,5.084,148.941
C07037=1109.430,-73.425,-48.321,179.774,5.080,148.940
C07038=1109.434,-73.640,-48.311,179.775,5.076,148.939
C07039=1109.440,-73.890,-48.301,179.774,5.070,148.938
C07040=1109.445,-74.139,-48.289,179.774,5.065,148.937
C07041=1109.450,-74.389,-48.279,179.775,5.060,148.936
C07042=1109.456,-74.639,-48.267,179.775,5.055,148.934
C07043=1109.461,-74.889,-48.257,179.775,5.050,148.933
C07044=1109.466,-75.138,-48.246,179.775,5.045,148.932
C07045=1109.471,-75.388,-48.235,179.775,5.039,148.931
C07046=1109.476,-75.638,-48.223,179.775,5.034,148.930
C07047=1109.482,-75.887,-48.212,179.775,5.029,148.929
C07048=1109.487,-76.137,-48.202,179.776,5.024,148.927
C07049=1109.492,-76.387,-48.192,179.776,5.019,148.926
C07050=1109.497,-76.636,-48.180,179.776,5.014,148.925
C07051=1109.503,-76.886,-48.169,179.776,5.009,148.924
C07052=1109.508,-77.136,-48.158,179.776,5.003,148.923
C07053=1109.513,-77.386,-48.148,179.776,4.998,148.922
C07054=1109.518,-77.635,-48.137,179.776,4.993,148.920
C07055=1109.523,-77.885,-48.126,179.777,4.988,148.919
C07056=1109.529,-78.134,-48.115,179.777,4.983,148.918
C07057=1109.534,-78.385,-48.104,179.777,4.978,148.917
C07058=1109.540,-78.634,-48.093,179.777,4.973,148.916
C07059=1109.545,-78.884,-48.082,179.777,4.967,148.914
C07060=1109.550,-79.133,-48.072,179.777,4.962,148.913
C07061=1109.555,-79.383,-48.061,179.778,4.957,148.912
C07062=1109.561,-79.633,-48.051,179.778,4.952,148.911
C07063=1109.566,-79.883,-48.040,179.778,4.947,148.910
C07064=1109.570,-80.133,-48.029,179.778,4.942,148.909
C07065=1109.577,-80.382,-48.018,179.778,4.937,148.907
C07066=1109.581,-80.632,-48.007,179.778,4.931,148.906
C07067=1109.587,-80.882,-47.997,179.779,4.926,148.905
C07068=1109.592,-81.132,-47.986,179.779,4.922,148.904
C07069=1109.597,-81.381,-47.975,179.779,4.917,148.903
C07070=1109.602,-81.631,-47.965,179.780,4.912,148.902
C07071=1109.608,-81.880,-47.954,179.780,4.906,148.900
C07072=1109.612,-82.130,-47.943,179.780,4.901,148.899
C07073=1109.618,-82.380,-47.933,179.781,4.896,148.898
C07074=1109.623,-82.630,-47.922,179.781,4.891,148.897
C07075=1109.629,-82.879,-47.912,179.781,4.886,148.895
C07076=1109.633,-83.129,-47.901,179.781,4.880,148.894
C07077=1109.639,-83.379,-47.891,179.781,4.875,148.893
C07078=1109.645,-83.628,-47.880,179.782,4.871,148.892
C07079=1109.650,-83.878,-47.870,179.782,4.866,148.891
C07080=1109.655,-84.127,-47.859,179.782,4.861,148.890
C07081=1109.660,-84.378,-47.848,179.783,4.855,148.888
C07082=1109.665,-84.627,-47.838,179.783,4.850,148.887
C07083=1109.670,-84.877,-47.827,179.783,4.845,148.886
C07084=1109.676,-85.126,-47.817,179.784,4.840,148.885
C07085=1109.681,-85.377,-47.806,179.784,4.835,148.883
C07086=1109.686,-85.626,-47.796,179.785,4.830,148.882
C07087=1109.691,-85.842,-47.786,179.784,4.825,148.881
C07088=1109.695,-86.055,-47.777,179.785,4.821,148.880
C07089=1109.700,-86.270,-47.768,179.785,4.817,148.879
C07090=1109.704,-86.485,-47.760,179.786,4.813,148.878
C07091=1109.709,-86.700,-47.750,179.786,4.808,148.877
C07092=1109.713,-86.915,-47.741,179.787,4.804,148.876
C07093=1109.718,-87.129,-47.733,179.787,4.800,148.875
C07094=1109.722,-87.345,-47.724,179.787,4.796,148.874
C07095=1109.728,-87.594,-47.713,179.787,4.791,148.873
C07096=1109.733,-87.843,-47.703,179.788,4.785,148.871
C07097=1109.738,-88.093,-47.692,179.788,4.780,148.870
C07098=1109.744,-88.343,-47.682,179.789,4.776,148.869
C07099=1109.749,-88.593,-47.671,179.789,4.770,148.868
C07100=1109.754,-88.842,-47.662,179.789,4.765,148.867
C07101=1109.759,-89.092,-47.652,179.789,4.760,148.865
C07102=1109.764,-89.342,-47.641,179.790,4.756,148.864
C07103=1109.770,-89.592,-47.631,179.790,4.751,148.863
C07104=1109.775,-89.842,-47.620,179.791,4.745,148.862
C07105=1109.780,-90.092,-47.610,179.792,4.741,148.860
C07106=1109.786,-90.340,-47.599,179.792,4.736,148.859
C07107=1109.791,-90.591,-47.588,179.792,4.730,148.858
C07108=1109.796,-90.840,-47.579,179.792,4.725,148.857
C07109=1109.801,-91.089,-47.569,179.793,4.721,148.856
C07110=1109.806,-91.340,-47.558,179.793,4.716,148.854
C07111=1109.812,-91.589,-47.548,179.794,4.711,148.853
C07112=1109.817,-91.839,-47.537,179.794,4.706,148.852
C07113=1109.822,-92.089,-47.527,179.795,4.701,148.851
C07114=1109.827,-92.338,-47.517,179.796,4.696,148.849
C07115=1109.832,-92.588,-47.507,179.796,4.691,148.848
C07116=1109.838,-92.838,-47.497,179.796,4.686,148.847
C07117=1109.843,-93.088,-47.486,179.797,4.682,148.846
C07118=1109.848,-93.338,-47.476,179.797,4.677,148.845
C07119=1109.854,-93.587,-47.466,179.797,4.672,148.844
C07120=1109.859,-93.837,-47.456,179.798,4.667,148.842
C07121=1109.864,-94.087,-47.446,179.798,4.662,148.841
C07122=1109.870,-94.337,-47.436,179.799,4.658,148.840
C07123=1109.875,-94.587,-47.426,179.799,4.653,148.839
C07124=1109.880,-94.836,-47.416,179.800,4.647,148.838
C07125=1109.885,-95.086,-47.406,179.800,4.643,148.836
C07126=1109.891,-95.336,-47.395,179.801,4.638,148.835
C07127=1109.896,-95.585,-47.385,179.801,4.633,148.834
C07128=1109.901,-95.835,-47.375,179.801,4.628,148.833
C07129=1109.906,-96.085,-47.365,179.802,4.623,148.832
C07130=1109.912,-96.334,-47.355,179.802,4.618,148.830
C07131=1109.917,-96.584,-47.344,179.802,4.613,148.829
C07132=1109.923,-96.835,-47.335,179.803,4.609,148.828
C07133=1109.928,-97.084,-47.325,179.803,4.603,148.827
C07134=1109.933,-97.333,-47.315,179.804,4.598,148.826
C07135=1109.938,-97.584,-47.304,179.804,4.593,148.824
C07136=1109.943,-97.833,-47.295,179.805,4.589,148.823
C07137=1109.949,-98.082,-47.285,179.805,4.584,148.822
C07138=1109.955,-98.333,-47.275,179.805,4.578,148.821
C07139=1109.960,-98.583,-47.264,179.806,4.574,148.820
C07140=1109.964,-98.832,-47.255,179.806,4.569,148.819
C07141=1109.970,-99.082,-47.245,179.806,4.564,148.817
C07142=1109.976,-99.331,-47.234,179.806,4.559,148.816
C07143=1109.980,-99.546,-47.226,179.807,4.555,148.815
C07144=1109.984,-99.761,-47.217,179.808,4.550,148.814
C07145=1109.989,-99.976,-47.210,179.808,4.546,148.813
C07146=1109.994,-100.191,-47.200,179.808,4.542,148.812
C07147=1109.998,-100.406,-47.192,179.808,4.538,148.811
C07148=1110.003,-100.620,-47.184,179.809,4.533,148.810
C07149=1110.008,-100.835,-47.175,179.809,4.529,148.809
C07150=1110.012,-101.050,-47.166,179.809,4.525,148.808
C07151=1110.017,-101.299,-47.157,179.809,4.520,148.807
C07152=1110.022,-101.550,-47.147,179.810,4.515,148.806
C07153=1110.028,-101.799,-47.137,179.810,4.510,148.804
C07154=1110.032,-102.049,-47.127,179.811,4.506,148.803
C07155=1110.038,-102.299,-47.117,179.811,4.500,148.802
C07156=1110.044,-102.549,-47.107,179.811,4.495,148.801
C07157=1110.049,-102.798,-47.098,179.811,4.490,148.800
C07158=1110.054,-103.048,-47.087,179.812,4.485,148.798
C07159=1110.059,-103.298,-47.078,179.812,4.481,148.797
C07160=1110.064,-103.548,-47.068,179.813,4.475,148.796
C07161=1110.069,-103.797,-47.058,179.813,4.470,148.795
C07162=1110.075,-104.047,-47.049,179.814,4.465,148.793
C07163=1110.081,-104.297,-47.039,179.814,4.460,148.792
C07164=1110.085,-104.546,-47.029,179.815,4.455,148.791
C07165=1110.091,-104.797,-47.019,179.815,4.450,148.790
C07166=1110.096,-105.046,-47.010,179.815,4.445,148.789
C07167=1110.101,-105.295,-46.999,179.815,4.440,148.787
C07168=1110.107,-105.545,-46.990,179.816,4.435,148.786
C07169=1110.112,-105.795,-46.980,179.816,4.430,148.785
C07170=1110.117,-106.045,-46.971,179.817,4.425,148.784
C07171=1110.122,-106.295,-46.961,179.817,4.420,148.783
C07172=1110.128,-106.545,-46.952,179.817,4.415,148.781
C07173=1110.133,-106.794,-46.942,179.818,4.411,148.780
C07174=1110.139,-107.044,-46.931,179.818,4.405,148.779
C07175=1110.144,-107.294,-46.923,179.818,4.400,148.778
C07176=1110.149,-107.543,-46.912,179.819,4.395,148.777
C07177=1110.155,-107.793,-46.903,179.819,4.390,148.775
C07178=1110.160,-108.043,-46.893,179.819,4.385,148.774
C07179=1110.165,-108.293,-46.884,179.820,4.380,148.773
C07180=1110.170,-108.542,-46.874,179.820,4.375,148.772
C07181=1110.176,-108.793,-46.865,179.821,4.370,148.771
C07182=1110.180,-109.042,-46.855,179.821,4.365,148.769
C07183=1110.186,-109.292,-46.846,179.822,4.359,148.768
C07184=1110.191,-109.541,-46.836,179.822,4.354,148.767
C07185=1110.197,-109.791,-46.827,179.823,4.350,148.765
C07186=1110.202,-110.041,-46.817,179.823,4.345,148.764
C07187=1110.207,-110.291,-46.807,179.823,4.340,148.763
C07188=1110.212,-110.541,-46.798,179.823,4.334,148.762
C07189=1110.218,-110.791,-46.788,179.824,4.329,148.761
C07190=1110.223,-111.040,-46.778,179.824,4.324,148.759
C07191=1110.228,-111.290,-46.770,179.824,4.319,148.758
C07192=1110.234,-111.540,-46.760,179.825,4.315,148.757
C07193=1110.239,-111.789,-46.750,179.826,4.309,148.756
C07194=1110.245,-112.040,-46.741,179.826,4.304,148.754
C07195=1110.250,-112.289,-46.731,179.826,4.299,148.753
C07196=1110.255,-112.539,-46.722,179.826,4.294,148.752
C07197=1110.261,-112.789,-46.713,179.827,4.288,148.751
C07198=1110.266,-113.038,-46.703,179.827,4.283,148.750
C07199=1110.270,-113.253,-46.696,179.828,4.279,148.748
C07200=1110.274,-113.468,-46.687,179.828,4.275,148.747
C07201=1110.279,-113.683,-46.679,179.828,4.270,148.746
C07202=1110.284,-113.898,-46.671,179.829,4.266,148.745
C07203=1110.288,-114.113,-46.663,179.829,4.262,148.744
C07204=1110.293,-114.327,-46.655,179.829,4.257,148.743
C07205=1110.298,-114.542,-46.648,179.830,4.253,148.742
C07206=1110.302,-114.757,-46.639,179.830,4.248,148.741
C07207=1110.308,-115.007,-46.630,179.831,4.243,148.740
C07208=1110.312,-115.257,-46.620,179.831,4.238,148.738
C07209=1110.318,-115.507,-46.611,179.831,4.233,148.737
C07210=1110.323,-115.757,-46.601,179.832,4.228,148.736
C07211=1110.329,-116.006,-46.592,179.832,4.222,148.735
C07212=1110.334,-116.255,-46.583,179.833,4.217,148.733
C07213=1110.340,-116.506,-46.574,179.833,4.212,148.732
C07214=1110.345,-116.755,-46.565,179.833,4.207,148.731
C07215=1110.350,-117.005,-46.555,179.833,4.202,148.730
C07216=1110.356,-117.255,-46.546,179.834,4.196,148.728
C07217=1110.361,-117.505,-46.537,179.835,4.191,148.727
C07218=1110.366,-117.755,-46.528,179.835,4.186,148.726
C07219=1110.372,-118.005,-46.518,179.835,4.181,148.725
C07220=1110.377,-118.254,-46.509,179.835,4.175,148.723
C07221=1110.382,-118.504,-46.500,179.836,4.170,148.722
C07222=1110.387,-118.754,-46.491,179.836,4.165,148.721
C07223=1110.393,-119.004,-46.481,179.837,4.160,148.720
C07224=1110.398,-119.254,-46.473,179.837,4.154,148.718
C07225=1110.403,-119.503,-46.463,179.838,4.149,148.717
C07226=1110.408,-119.753,-46.454,179.838,4.144,148.716
C07227=1110.414,-120.003,-46.445,179.838,4.138,148.714
C07228=1110.420,-120.253,-46.436,179.839,4.133,148.713
C07229=1110.425,-120.503,-46.427,179.839,4.128,148.712
C07230=1110.430,-120.752,-46.418,179.840,4.123,148.711
C07231=1110.435,-121.002,-46.408,179.840,4.117,148.709
C07232=1110.441,-121.252,-46.399,179.841,4.112,148.708
C07233=1110.446,-121.501,-46.390,179.841,4.107,148.707
C07234=1110.452,-121.751,-46.381,179.841,4.102,148.705
C07235=1110.457,-122.001,-46.372,179.842,4.096,148.704
C07236=1110.462,-122.251,-46.364,179.842,4.091,148.703
C07237=1110.467,-122.500,-46.355,179.843,4.086,148.702
C07238=1110.473,-122.751,-46.345,179.843,4.081,148.700
C07239=1110.478,-123.000,-46.336,179.844,4.075,148.699
C07240=1110.483,-123.250,-46.327,179.844,4.070,148.698
C07241=1110.488,-123.500,-46.318,179.844,4.065,148.696
C07242=1110.494,-123.749,-46.310,179.845,4.059,148.695
C07243=1110.499,-123.998,-46.300,179.846,4.054,148.694
C07244=1110.505,-124.249,-46.291,179.846,4.049,148.693
C07245=1110.510,-124.499,-46.282,179.847,4.043,148.691
C07246=1110.515,-124.748,-46.273,179.847,4.038,148.690
C07247=1110.520,-124.998,-46.264,179.848,4.033,148.688
C07248=1110.526,-125.248,-46.255,179.848,4.027,148.687
C07249=1110.531,-125.497,-46.247,179.848,4.022,148.686
C07250=1110.537,-125.747,-46.238,179.849,4.017,148.684
C07251=1110.542,-125.997,-46.229,179.849,4.011,148.683
C07252=1110.547,-126.247,-46.221,179.850,4.005,148.682
C07253=1110.552,-126.497,-46.212,179.850,4.000,148.681
C07254=1110.558,-126.747,-46.202,179.850,3.995,148.679
C07255=1110.562,-126.962,-46.195,179.851,3.990,148.678
C07256=1110.567,-127.177,-46.187,179.851,3.985,148.677
C07257=1110.572,-127.392,-46.179,179.852,3.981,148.676
C07258=1110.576,-127.607,-46.172,179.852,3.976,148.675
C07259=1110.581,-127.822,-46.165,179.852,3.971,148.673
C07260=1110.585,-128.037,-46.157,179.853,3.967,148.672
C07261=1110.590,-128.252,-46.150,179.853,3.962,148.671
C07262=1110.595,-128.467,-46.142,179.854,3.958,148.670
C07263=1110.172,-128.457,-46.167,179.861,3.961,148.669
C07264=1110.167,-128.242,-46.175,179.861,3.966,148.670
C07265=1110.162,-128.027,-46.183,179.861,3.971,148.671
C07266=1110.158,-127.812,-46.191,179.860,3.976,148.672
C07267=1110.154,-127.598,-46.198,179.860,3.980,148.673
C07268=1110.149,-127.383,-46.206,179.859,3.985,148.674
C07269=1110.144,-127.167,-46.213,179.859,3.990,148.676
C07270=1110.139,-126.952,-46.221,179.858,3.994,148.677
C07271=1110.135,-126.737,-46.229,179.858,3.999,148.678
C07272=1110.129,-126.487,-46.237,179.857,4.005,148.679
C07273=1110.124,-126.238,-46.246,179.857,4.010,148.681
C07274=1110.119,-125.988,-46.255,179.857,4.015,148.682
C07275=1110.114,-125.738,-46.264,179.856,4.020,148.683
C07276=1110.108,-125.489,-46.273,179.855,4.026,148.684
C07277=1110.103,-125.239,-46.282,179.855,4.031,148.686
C07278=1110.098,-124.989,-46.290,179.854,4.036,148.687
C07279=1110.092,-124.739,-46.300,179.854,4.042,148.688
C07280=1110.087,-124.489,-46.309,179.854,4.048,148.690
C07281=1110.082,-124.239,-46.318,179.854,4.053,148.691
C07282=1110.076,-123.989,-46.327,179.853,4.059,148.693
C07283=1110.072,-123.740,-46.336,179.852,4.064,148.694
C07284=1110.066,-123.491,-46.345,179.852,4.069,148.695
C07285=1110.061,-123.241,-46.354,179.851,4.074,148.696
C07286=1110.055,-122.991,-46.363,179.851,4.080,148.698
C07287=1110.050,-122.741,-46.372,179.851,4.085,148.699
C07288=1110.044,-122.491,-46.381,179.850,4.090,148.700
C07289=1110.039,-122.241,-46.390,179.850,4.096,148.702
C07290=1110.034,-121.991,-46.399,179.849,4.101,148.703
C07291=1110.028,-121.741,-46.408,179.849,4.106,148.704
C07292=1110.023,-121.491,-46.417,179.848,4.111,148.705
C07293=1110.018,-121.242,-46.427,179.848,4.117,148.707
C07294=1110.013,-120.992,-46.436,179.848,4.122,148.708
C07295=1110.007,-120.743,-46.444,179.847,4.127,148.709
C07296=1110.001,-120.493,-46.454,179.847,4.132,148.711
C07297=1109.996,-120.243,-46.463,179.846,4.138,148.712
C07298=1109.991,-119.993,-46.471,179.846,4.143,148.713
C07299=1109.986,-119.744,-46.481,179.845,4.148,148.714
C07300=1109.980,-119.494,-46.491,179.845,4.153,148.716
C07301=1109.975,-119.244,-46.499,179.845,4.159,148.717
C07302=1109.970,-118.994,-46.508,179.844,4.164,148.718
C07303=1109.965,-118.744,-46.517,179.844,4.169,148.720
C07304=1109.959,-118.495,-46.527,179.843,4.174,148.721
C07305=1109.954,-118.245,-46.536,179.843,4.180,148.722
C07306=1109.949,-117.995,-46.545,179.842,4.185,148.723
C07307=1109.943,-117.745,-46.555,179.842,4.190,148.725
C07308=1109.938,-117.496,-46.564,179.842,4.195,148.726
C07309=1109.933,-117.246,-46.573,179.841,4.201,148.727
C07310=1109.927,-116.996,-46.583,179.840,4.205,148.729
C07311=1109.922,-116.746,-46.592,179.840,4.211,148.730
C07312=1109.917,-116.497,-46.601,179.840,4.216,148.731
C07313=1109.912,-116.247,-46.610,179.839,4.221,148.732
C07314=1109.906,-115.997,-46.620,179.839,4.226,148.733
C07315=1109.901,-115.747,-46.629,179.838,4.232,148.735
C07316=1109.895,-115.497,-46.639,179.838,4.237,148.736
C07317=1109.890,-115.247,-46.648,179.838,4.242,148.737
C07318=1109.885,-114.998,-46.657,179.837,4.247,148.738
C07319=1109.879,-114.748,-46.667,179.837,4.252,148.740
C07320=1109.875,-114.534,-46.675,179.836,4.257,148.741
C07321=1109.870,-114.318,-46.683,179.836,4.261,148.742
C07322=1109.865,-114.104,-46.691,179.836,4.266,148.743
C07323=1109.861,-113.888,-46.699,179.835,4.270,148.744
C07324=1109.857,-113.674,-46.707,179.836,4.274,148.745
C07325=1109.852,-113.459,-46.715,179.835,4.279,148.746
C07326=1109.847,-113.244,-46.723,179.834,4.283,148.747
C07327=1109.842,-113.029,-46.731,179.834,4.288,148.748
C07328=1109.838,-112.780,-46.741,179.833,4.292,148.750
C07329=1109.832,-112.530,-46.750,179.833,4.297,148.751
C07330=1109.827,-112.280,-46.760,179.833,4.303,148.752
C07331=1109.821,-112.030,-46.769,179.833,4.308,148.753
C07332=1109.817,-111.780,-46.779,179.832,4.313,148.754
C07333=1109.811,-111.530,-46.788,179.832,4.318,148.756
C07334=1109.806,-111.280,-46.798,179.831,4.324,148.757
C07335=1109.801,-111.031,-46.807,179.831,4.329,148.758
C07336=1109.795,-110.781,-46.817,179.830,4.333,148.759
C07337=1109.790,-110.532,-46.826,179.830,4.338,148.761
C07338=1109.784,-110.282,-46.836,179.830,4.343,148.762
C07339=1109.779,-110.032,-46.845,179.829,4.349,148.763
C07340=1109.773,-109.782,-46.855,179.829,4.354,148.764
C07341=1109.768,-109.533,-46.864,179.829,4.359,148.765
C07342=1109.763,-109.283,-46.873,179.828,4.363,148.767
C07343=1109.758,-109.033,-46.884,179.828,4.368,148.768
C07344=1109.753,-108.783,-46.893,179.827,4.374,148.769
C07345=1109.747,-108.533,-46.903,179.827,4.379,148.771
C07346=1109.742,-108.284,-46.912,179.827,4.384,148.772
C07347=1109.737,-108.034,-46.922,179.826,4.389,148.773
C07348=1109.732,-107.785,-46.932,179.826,4.394,148.774
C07349=1109.726,-107.535,-46.941,179.825,4.399,148.775
C07350=1109.721,-107.284,-46.952,179.825,4.404,148.777
C07351=1109.716,-107.035,-46.961,179.825,4.409,148.778
C07352=1109.710,-106.785,-46.971,179.825,4.414,148.779
C07353=1109.705,-106.535,-46.980,179.824,4.419,148.780
C07354=1109.699,-106.286,-46.990,179.824,4.424,148.781
C07355=1109.695,-106.036,-47.000,179.823,4.429,148.783
C07356=1109.689,-105.786,-47.009,179.823,4.434,148.784
C07357=1109.684,-105.536,-47.019,179.823,4.439,148.785
C07358=1109.679,-105.287,-47.029,179.822,4.444,148.786
C07359=1109.674,-105.037,-47.038,179.822,4.449,148.787
C07360=1109.668,-104.787,-47.048,179.822,4.454,148.789
C07361=1109.662,-104.538,-47.059,179.821,4.459,148.790
C07362=1109.658,-104.287,-47.068,179.821,4.465,148.791
C07363=1109.652,-104.038,-47.078,179.820,4.469,148.792
C07364=1109.647,-103.788,-47.088,179.820,4.474,148.794
C07365=1109.642,-103.538,-47.097,179.819,4.479,148.795
C07366=1109.636,-103.289,-47.107,179.819,4.484,148.796
C07367=1109.632,-103.039,-47.117,179.818,4.489,148.797
C07368=1109.626,-102.789,-47.127,179.818,4.494,148.798
C07369=1109.621,-102.539,-47.137,179.818,4.499,148.800
C07370=1109.615,-102.290,-47.147,179.818,4.504,148.801
C07371=1109.610,-102.040,-47.157,179.817,4.509,148.802
C07372=1109.605,-101.790,-47.166,179.817,4.514,148.803
C07373=1109.600,-101.540,-47.176,179.816,4.519,148.804
C07374=1109.594,-101.291,-47.187,179.816,4.524,148.806
C07375=1109.589,-101.041,-47.196,179.816,4.529,148.807
